Yaskawa INFORM job: pointsclTRJ4.JBI

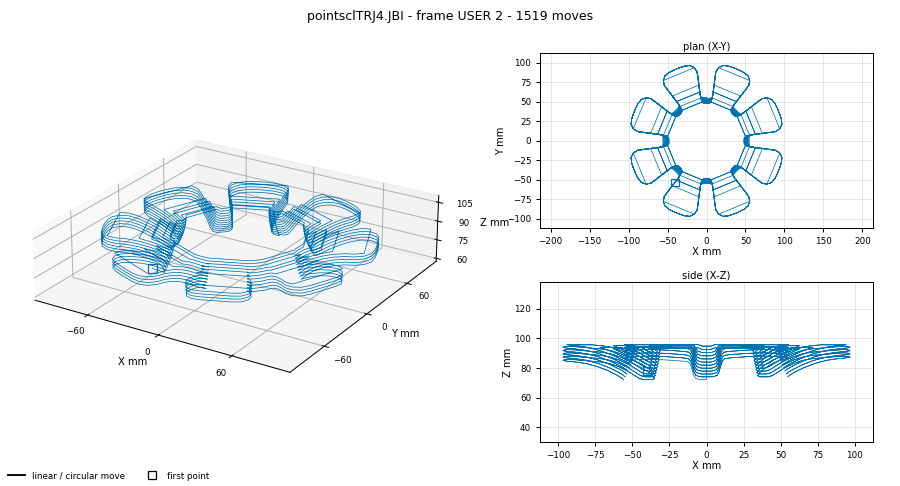
[picture p0: tool path of pointsclTRJ4.JBI in frame USER 2, 1519 of 1519 moves have a stored position in this frame; points joined in program order, loops and branches not executed]
/JOB
//NAME pointsclTRJ4
//POS
///NPOS 1519,0,0,0,0,0
///USER 2
///TOOL 1
///POSTYPE USER
///RECTAN
///RCONF 1,0,0,0,0,0,0,0,0,0,0,0,0,0,0,0,0,0,0,0,0,0,0,0
C00000=-40.007,-53.324,78.036,162.0773,27.0568,0.0000
C00001=-36.517,-48.718,75.143,159.1189,26.0241,0.0000
C00002=-35.037,-45.351,73.015,156.9441,24.9731,0.0000
C00003=-36.538,-42.505,72.166,153.8641,22.7812,0.0000
C00004=-38.303,-40.803,72.129,153.4120,22.4132,0.0000
C00005=-39.567,-39.567,72.154,154.3066,23.4380,0.0000
C00006=-40.803,-38.303,72.129,155.2410,24.4422,0.0000
C00007=-42.506,-36.538,72.166,154.9286,23.9614,0.0000
C00008=-45.352,-35.037,73.015,153.1527,20.7940,0.0000
C00009=-48.718,-36.517,75.143,152.4095,18.6805,0.0000
C00010=-53.324,-40.007,78.036,151.7719,15.9057,0.0000
C00011=-59.196,-44.618,80.927,152.7519,8.2885,0.0000
C00012=-65.578,-49.604,83.062,-179.3107,0.4201,0.0000
C00013=-71.524,-53.949,84.088,-176.3228,2.4871,0.0000
C00014=-77.795,-55.184,84.621,-175.2384,3.2785,0.0000
C00015=-83.601,-53.037,85.050,-174.7144,3.6343,0.0000
C00016=-87.741,-47.957,85.481,-174.6375,3.6773,0.0000
C00017=-90.934,-41.602,85.762,-174.7812,3.5713,0.0000
C00018=-93.717,-34.883,85.762,173.7849,-1.1544,0.0000
C00019=-95.953,-28.131,85.481,173.6084,-1.1802,0.0000
C00020=-96.617,-21.612,85.050,173.6932,-1.1566,0.0000
C00021=-94.030,-15.989,84.621,174.3152,-1.0407,0.0000
C00022=-88.723,-12.427,84.088,175.6413,-0.8379,0.0000
C00023=-81.446,-11.295,83.062,179.2156,-0.1904,0.0000
C00024=-73.408,-10.308,80.927,-166.0561,24.9794,0.0000
C00025=-65.995,-9.417,78.036,-171.4191,31.0262,0.0000
C00026=-60.270,-8.627,75.143,-174.3026,32.4608,0.0000
C00027=-56.844,-7.293,73.015,-176.7405,33.3374,0.0000
C00028=-55.892,-4.219,72.166,179.0738,34.1239,0.0000
C00029=-55.936,-1.768,72.129,178.4088,34.2068,0.0000
C00030=-55.957,0.000,72.154,179.9988,34.2310,0.0000
C00031=-55.936,1.767,72.129,-178.4074,34.2068,0.0000
C00032=-55.892,4.220,72.166,-179.0753,34.1238,0.0000
C00033=-56.844,7.293,73.015,176.7400,33.3374,0.0000
C00034=-60.270,8.627,75.143,174.3025,32.4608,0.0000
C00035=-65.995,9.417,78.036,171.4191,31.0263,0.0000
C00036=-73.408,10.308,80.927,166.0562,24.9798,0.0000
C00037=-81.446,11.295,83.062,-179.2156,-0.1904,0.0000
C00038=-88.723,12.427,84.088,-175.6413,-0.8379,0.0000
C00039=-94.030,15.989,84.621,-174.3152,-1.0407,0.0000
C00040=-96.617,21.612,85.050,-173.6932,-1.1566,0.0000
C00041=-95.953,28.131,85.481,-173.6084,-1.1802,0.0000
C00042=-93.717,34.883,85.762,-173.7849,-1.1544,0.0000
C00043=-90.934,41.602,85.762,174.7812,3.5713,0.0000
C00044=-87.741,47.957,85.481,174.6375,3.6773,0.0000
C00045=-83.601,53.037,85.050,174.7144,3.6343,0.0000
C00046=-77.795,55.184,84.621,175.2384,3.2785,0.0000
C00047=-71.524,53.949,84.088,176.3228,2.4871,0.0000
C00048=-65.578,49.604,83.062,179.3107,0.4201,0.0000
C00049=-59.196,44.618,80.927,-152.7521,8.2881,0.0000
C00050=-53.324,40.007,78.036,-151.7719,15.9056,0.0000
C00051=-48.718,36.517,75.143,-152.4095,18.6805,0.0000
C00052=-45.351,35.037,73.015,-153.1530,20.7943,0.0000
C00053=-42.505,36.538,72.166,-154.9295,23.9624,0.0000
C00054=-40.803,38.303,72.129,-155.2402,24.4413,0.0000
C00055=-39.567,39.567,72.154,-154.3081,23.4396,0.0000
C00056=-38.303,40.803,72.129,-153.4112,22.4123,0.0000
C00057=-36.538,42.506,72.166,-153.8651,22.7821,0.0000
C00058=-35.037,45.352,73.015,-156.9444,24.9734,0.0000
C00059=-36.517,48.718,75.143,-159.1190,26.0242,0.0000
C00060=-40.007,53.324,78.036,-162.0772,27.0569,0.0000
C00061=-44.618,59.196,80.927,-170.6940,26.9403,0.0000
C00062=-49.604,65.578,83.062,-179.5799,-0.6893,0.0000
C00063=-53.949,71.524,84.088,-177.5078,-3.6738,0.0000
C00064=-55.184,77.795,84.621,-176.7102,-4.7538,0.0000
C00065=-53.037,83.601,85.050,-176.3502,-5.2749,0.0000
C00066=-47.957,87.741,85.481,-176.3066,-5.3514,0.0000
C00067=-41.602,90.934,85.762,-176.4139,-5.2087,0.0000
C00068=-34.883,93.717,85.762,178.8388,6.2138,0.0000
C00069=-28.131,95.953,85.481,178.8125,6.3902,0.0000
C00070=-21.612,96.617,85.050,178.8363,6.3055,0.0000
C00071=-15.989,94.030,84.621,178.9542,5.6839,0.0000
C00072=-12.427,88.723,84.088,179.1597,4.3583,0.0000
C00073=-11.295,81.446,83.062,179.8096,0.7844,0.0000
C00074=-10.308,73.408,80.927,-154.3579,-12.6167,0.0000
C00075=-9.417,65.995,78.036,-148.6881,-7.3459,0.0000
C00076=-8.627,60.270,75.143,-147.4105,-4.8050,0.0000
C00077=-7.293,56.844,73.015,-146.6200,-2.7231,0.0000
C00078=-4.220,55.892,72.166,-145.8728,0.7655,0.0000
C00079=-1.767,55.936,72.129,-145.7829,1.3171,0.0000
C00080=0.000,55.957,72.154,-145.7690,-0.0010,0.0000
C00081=0.000,54.840,74.049,-146.5029,-0.0011,0.0000
C00082=1.666,54.823,74.024,-146.5152,-1.2504,0.0000
C00083=4.048,54.790,74.062,-146.6018,-0.7445,0.0000
C00084=7.088,55.804,74.943,-147.3459,2.7005,0.0000
C00085=8.393,59.388,77.145,-148.1466,4.7745,0.0000
C00086=9.180,65.335,80.122,-149.5349,7.4435,0.0000
C00087=10.089,72.980,83.074,-156.5768,13.0945,0.0000
C00088=11.094,81.206,85.240,179.6071,-1.7912,0.0000
C00089=12.226,88.613,86.276,179.1566,-4.6034,0.0000
C00090=15.808,94.009,86.813,178.9836,-5.7439,0.0000
C00091=21.475,96.642,87.246,178.8772,-6.3083,0.0000
C00092=28.048,95.980,87.679,178.8549,-6.3901,0.0000
C00093=34.856,93.728,87.962,178.8775,-6.2344,0.0000
C00094=41.629,90.922,87.962,-176.3720,5.1958,0.0000
C00095=48.035,87.701,87.679,-176.2769,5.3214,0.0000
C00096=53.151,83.521,87.246,-176.3195,5.2481,0.0000
C00097=55.296,77.652,86.813,-176.6467,4.7753,0.0000
C00098=54.014,71.304,86.276,-177.3359,3.8489,0.0000
C00099=49.577,65.266,85.240,-179.0109,1.5443,0.0000
C00100=44.470,58.738,83.074,-172.7574,-25.7204,0.0000
C00101=39.708,52.690,80.122,-162.8416,-26.5576,0.0000
C00102=36.059,47.928,77.145,-159.7054,-25.5142,0.0000
C00103=34.447,44.472,74.943,-157.5329,-24.4829,0.0000
C00104=35.880,41.605,74.062,-154.4883,-22.3343,0.0000
C00105=37.588,39.944,74.024,-154.0682,-21.9995,0.0000
C00106=38.778,38.778,74.049,-154.9210,-22.9691,0.0000
C00107=39.943,37.588,74.024,-155.8089,-23.9209,0.0000
C00108=41.605,35.880,74.062,-155.5235,-23.4763,0.0000
C00109=44.472,34.447,74.943,-153.7672,-20.3520,0.0000
C00110=47.928,36.059,77.145,-153.0297,-18.2415,0.0000
C00111=52.690,39.708,80.122,-152.3850,-15.3009,0.0000
C00112=58.738,44.470,83.074,-154.0994,-6.5221,0.0000
C00113=65.266,49.577,85.240,178.4555,-0.9887,0.0000
C00114=71.304,54.014,86.276,176.1470,-2.6581,0.0000
C00115=77.652,55.296,86.813,175.2165,-3.3416,0.0000
C00116=83.521,53.151,87.246,174.7411,-3.6651,0.0000
C00117=87.701,48.035,87.679,174.6674,-3.7070,0.0000
C00118=90.922,41.629,87.962,174.7939,-3.6131,0.0000
C00119=93.728,34.856,87.962,-173.7644,1.1158,0.0000
C00120=95.980,28.048,87.679,-173.6087,1.1380,0.0000
C00121=96.642,21.475,87.246,-173.6905,1.1160,0.0000
C00122=94.009,15.808,86.813,-174.2552,1.0113,0.0000
C00123=88.613,12.226,86.276,-175.3961,0.8406,0.0000
C00124=81.206,11.094,85.240,-178.2088,0.3927,0.0000
C00125=72.980,10.089,83.074,165.7755,-22.7793,0.0000
C00126=65.335,9.180,80.122,171.3809,-30.1815,0.0000
C00127=59.388,8.393,77.145,174.3839,-31.7299,0.0000
C00128=55.804,7.088,74.943,176.7935,-32.6133,0.0000
C00129=54.790,4.048,74.062,-179.1083,-33.3950,0.0000
C00130=54.823,1.666,74.024,-178.5009,-33.4758,0.0000
C00131=54.840,0.000,74.049,-179.9987,-33.4971,0.0000
C00132=54.823,-1.665,74.024,178.4994,-33.4758,0.0000
C00133=54.790,-4.048,74.062,179.1098,-33.3950,0.0000
C00134=55.804,-7.088,74.943,-176.7931,-32.6133,0.0000
C00135=59.388,-8.393,77.145,-174.3838,-31.7300,0.0000
C00136=65.335,-9.180,80.122,-171.3809,-30.1816,0.0000
C00137=72.980,-10.089,83.074,-165.7756,-22.7798,0.0000
C00138=81.206,-11.094,85.240,178.2088,0.3927,0.0000
C00139=88.613,-12.226,86.276,175.3961,0.8406,0.0000
C00140=94.009,-15.808,86.813,174.2552,1.0113,0.0000
C00141=96.642,-21.475,87.246,173.6905,1.1160,0.0000
C00142=95.980,-28.048,87.679,173.6087,1.1380,0.0000
C00143=93.728,-34.856,87.962,173.7644,1.1158,0.0000
C00144=90.922,-41.629,87.962,-174.7939,-3.6131,0.0000
C00145=87.701,-48.035,87.679,-174.6674,-3.7070,0.0000
C00146=83.521,-53.151,87.246,-174.7411,-3.6651,0.0000
C00147=77.652,-55.296,86.813,-175.2165,-3.3416,0.0000
C00148=71.304,-54.014,86.276,-176.1470,-2.6581,0.0000
C00149=65.266,-49.577,85.240,-178.4555,-0.9887,0.0000
C00150=58.738,-44.470,83.074,154.0997,-6.5217,0.0000
C00151=52.690,-39.708,80.122,152.3851,-15.3008,0.0000
C00152=47.928,-36.059,77.145,153.0298,-18.2415,0.0000
C00153=44.472,-34.447,74.943,153.7674,-20.3523,0.0000
C00154=41.605,-35.880,74.062,155.5243,-23.4773,0.0000
C00155=39.944,-37.588,74.024,155.8080,-23.9200,0.0000
C00156=38.778,-38.778,74.049,154.9225,-22.9708,0.0000
C00157=37.588,-39.943,74.024,154.0673,-21.9986,0.0000
C00158=35.880,-41.605,74.062,154.4893,-22.3352,0.0000
C00159=34.447,-44.472,74.943,157.5332,-24.4832,0.0000
C00160=36.059,-47.928,77.145,159.7054,-25.5143,0.0000
C00161=39.708,-52.690,80.122,162.8414,-26.5576,0.0000
C00162=44.470,-58.738,83.074,172.7569,-25.7206,0.0000
C00163=49.577,-65.266,85.240,179.0109,1.5443,0.0000
C00164=54.014,-71.304,86.276,177.3359,3.8489,0.0000
C00165=55.296,-77.652,86.813,176.6467,4.7753,0.0000
C00166=53.151,-83.521,87.246,176.3195,5.2481,0.0000
C00167=48.035,-87.701,87.679,176.2769,5.3214,0.0000
C00168=41.629,-90.922,87.962,176.3720,5.1958,0.0000
C00169=34.856,-93.728,87.962,-178.8775,-6.2344,0.0000
C00170=28.048,-95.980,87.679,-178.8549,-6.3901,0.0000
C00171=21.475,-96.642,87.246,-178.8772,-6.3083,0.0000
C00172=15.808,-94.009,86.813,-178.9836,-5.7439,0.0000
C00173=12.226,-88.613,86.276,-179.1566,-4.6034,0.0000
C00174=11.094,-81.206,85.240,-179.6071,-1.7912,0.0000
C00175=10.089,-72.980,83.074,156.5768,13.0945,0.0000
C00176=9.180,-65.335,80.122,149.5349,7.4435,0.0000
C00177=8.393,-59.388,77.145,148.1466,4.7745,0.0000
C00178=7.088,-55.804,74.943,147.3459,2.7005,0.0000
C00179=4.048,-54.790,74.062,146.6018,-0.7445,0.0000
C00180=1.666,-54.823,74.024,146.5152,-1.2504,0.0000
C00181=0.000,-54.840,74.049,146.5029,-0.0011,0.0000
C00182=0.000,-54.840,74.049,146.5029,-0.0011,0.0000
C00183=-1.665,-54.823,74.024,146.5152,1.2517,0.0000
C00184=-4.048,-54.790,74.062,146.6019,0.7432,0.0000
C00185=-7.088,-55.804,74.943,147.3460,-2.7009,0.0000
C00186=-8.393,-59.388,77.145,148.1466,-4.7746,0.0000
C00187=-9.180,-65.335,80.122,149.5348,-7.4435,0.0000
C00188=-10.089,-72.980,83.074,156.5763,-13.0943,0.0000
C00189=-11.094,-81.206,85.240,-179.6071,1.7912,0.0000
C00190=-12.226,-88.613,86.276,-179.1566,4.6034,0.0000
C00191=-15.808,-94.009,86.813,-178.9836,5.7439,0.0000
C00192=-21.475,-96.642,87.246,-178.8772,6.3083,0.0000
C00193=-28.048,-95.980,87.679,-178.8549,6.3901,0.0000
C00194=-34.856,-93.728,87.962,-178.8775,6.2344,0.0000
C00195=-41.629,-90.922,87.962,176.3720,-5.1958,0.0000
C00196=-48.035,-87.701,87.679,176.2769,-5.3214,0.0000
C00197=-53.151,-83.521,87.246,176.3195,-5.2481,0.0000
C00198=-55.296,-77.652,86.813,176.6467,-4.7753,0.0000
C00199=-54.014,-71.304,86.276,177.3359,-3.8489,0.0000
C00200=-49.577,-65.266,85.240,179.0109,-1.5443,0.0000
C00201=-44.470,-58.738,83.074,172.7574,25.7204,0.0000
C00202=-39.708,-52.690,80.122,162.8416,26.5576,0.0000
C00203=-36.059,-47.928,77.145,159.7054,25.5142,0.0000
C00204=-34.447,-44.472,74.943,157.5329,24.4829,0.0000
C00205=-35.880,-41.605,74.062,154.4883,22.3343,0.0000
C00206=-37.588,-39.944,74.024,154.0682,21.9995,0.0000
C00207=-38.778,-38.778,74.049,154.9210,22.9691,0.0000
C00208=-39.943,-37.588,74.024,155.8089,23.9209,0.0000
C00209=-41.605,-35.880,74.062,155.5235,23.4763,0.0000
C00210=-44.472,-34.447,74.943,153.7672,20.3520,0.0000
C00211=-47.928,-36.059,77.145,153.0297,18.2415,0.0000
C00212=-52.690,-39.708,80.122,152.3850,15.3009,0.0000
C00213=-58.738,-44.470,83.074,154.0994,6.5221,0.0000
C00214=-65.266,-49.577,85.240,-178.4555,0.9887,0.0000
C00215=-71.304,-54.014,86.276,-176.1470,2.6581,0.0000
C00216=-77.652,-55.296,86.813,-175.2165,3.3416,0.0000
C00217=-83.521,-53.151,87.246,-174.7411,3.6651,0.0000
C00218=-87.701,-48.035,87.679,-174.6674,3.7070,0.0000
C00219=-90.922,-41.629,87.962,-174.7939,3.6131,0.0000
C00220=-93.728,-34.856,87.962,173.7644,-1.1158,0.0000
C00221=-95.980,-28.048,87.679,173.6087,-1.1380,0.0000
C00222=-96.642,-21.475,87.246,173.6905,-1.1160,0.0000
C00223=-94.009,-15.808,86.813,174.2552,-1.0113,0.0000
C00224=-88.613,-12.226,86.276,175.3961,-0.8406,0.0000
C00225=-81.206,-11.094,85.240,178.2088,-0.3927,0.0000
C00226=-72.980,-10.089,83.074,-165.7755,22.7793,0.0000
C00227=-65.335,-9.180,80.122,-171.3809,30.1815,0.0000
C00228=-59.388,-8.393,77.145,-174.3839,31.7299,0.0000
C00229=-55.804,-7.088,74.943,-176.7935,32.6133,0.0000
C00230=-54.790,-4.048,74.062,179.1083,33.3950,0.0000
C00231=-54.823,-1.666,74.024,178.5009,33.4758,0.0000
C00232=-54.840,0.000,74.049,179.9987,33.4971,0.0000
C00233=-54.823,1.665,74.024,-178.4994,33.4758,0.0000
C00234=-54.790,4.048,74.062,-179.1098,33.3950,0.0000
C00235=-55.804,7.088,74.943,176.7931,32.6133,0.0000
C00236=-59.388,8.393,77.145,174.3838,31.7300,0.0000
C00237=-65.335,9.180,80.122,171.3809,30.1816,0.0000
C00238=-72.980,10.089,83.074,165.7756,22.7798,0.0000
C00239=-81.206,11.094,85.240,-178.2088,-0.3927,0.0000
C00240=-88.613,12.226,86.276,-175.3961,-0.8406,0.0000
C00241=-94.009,15.808,86.813,-174.2552,-1.0113,0.0000
C00242=-96.642,21.475,87.246,-173.6905,-1.1160,0.0000
C00243=-95.980,28.048,87.679,-173.6087,-1.1380,0.0000
C00244=-93.728,34.856,87.962,-173.7644,-1.1158,0.0000
C00245=-90.922,41.629,87.962,174.7939,3.6131,0.0000
C00246=-87.701,48.035,87.679,174.6674,3.7070,0.0000
C00247=-83.521,53.151,87.246,174.7411,3.6651,0.0000
C00248=-77.652,55.296,86.813,175.2165,3.3416,0.0000
C00249=-71.304,54.014,86.276,176.1470,2.6581,0.0000
C00250=-65.266,49.577,85.240,178.4555,0.9887,0.0000
C00251=-58.738,44.470,83.074,-154.0997,6.5217,0.0000
C00252=-52.690,39.708,80.122,-152.3851,15.3008,0.0000
C00253=-47.928,36.059,77.145,-153.0298,18.2415,0.0000
C00254=-44.472,34.447,74.943,-153.7674,20.3523,0.0000
C00255=-41.605,35.880,74.062,-155.5243,23.4773,0.0000
C00256=-39.944,37.588,74.024,-155.8080,23.9200,0.0000
C00257=-38.778,38.778,74.049,-154.9225,22.9708,0.0000
C00258=-37.588,39.943,74.024,-154.0673,21.9986,0.0000
C00259=-35.880,41.605,74.062,-154.4893,22.3352,0.0000
C00260=-34.447,44.472,74.943,-157.5332,24.4832,0.0000
C00261=-36.059,47.928,77.145,-159.7054,25.5143,0.0000
C00262=-39.708,52.690,80.122,-162.8414,26.5576,0.0000
C00263=-44.470,58.738,83.074,-172.7569,25.7206,0.0000
C00264=-49.577,65.266,85.240,-179.0109,-1.5443,0.0000
C00265=-54.014,71.304,86.276,-177.3359,-3.8489,0.0000
C00266=-55.296,77.652,86.813,-176.6467,-4.7753,0.0000
C00267=-53.151,83.521,87.246,-176.3195,-5.2481,0.0000
C00268=-48.035,87.701,87.679,-176.2769,-5.3214,0.0000
C00269=-41.629,90.922,87.962,-176.3720,-5.1958,0.0000
C00270=-34.856,93.728,87.962,178.8775,6.2344,0.0000
C00271=-28.048,95.980,87.679,178.8549,6.3901,0.0000
C00272=-21.475,96.642,87.246,178.8772,6.3083,0.0000
C00273=-15.808,94.009,86.813,178.9836,5.7439,0.0000
C00274=-12.226,88.613,86.276,179.1566,4.6034,0.0000
C00275=-11.094,81.206,85.240,179.6071,1.7912,0.0000
C00276=-10.089,72.980,83.074,-156.5763,-13.0943,0.0000
C00277=-9.180,65.335,80.122,-149.5348,-7.4435,0.0000
C00278=-8.393,59.388,77.145,-148.1466,-4.7746,0.0000
C00279=-7.088,55.804,74.943,-147.3460,-2.7009,0.0000
C00280=-4.048,54.790,74.062,-146.6019,0.7432,0.0000
C00281=-1.665,54.823,74.024,-146.5152,1.2517,0.0000
C00282=0.000,54.840,74.049,-146.5029,-0.0011,0.0000
C00283=0.000,53.776,75.975,-147.2942,-0.0011,0.0000
C00284=1.568,53.762,75.948,-147.3046,-1.1830,0.0000
C00285=3.884,53.739,75.988,-147.3883,-0.7211,0.0000
C00286=6.894,54.818,76.900,-148.1310,2.6757,0.0000
C00287=8.175,58.565,79.173,-148.9497,4.7476,0.0000
C00288=8.965,64.737,82.228,-150.4833,7.5652,0.0000
C00289=9.898,72.606,85.234,-159.4646,13.4583,0.0000
C00290=10.924,81.005,87.424,179.4966,-2.4962,0.0000
C00291=12.061,88.524,88.468,179.1698,-4.7418,0.0000
C00292=15.662,93.991,89.008,179.0218,-5.7312,0.0000
C00293=21.365,96.662,89.443,178.9256,-6.2465,0.0000
C00294=27.983,96.002,89.878,178.9048,-6.3264,0.0000
C00295=34.834,93.736,90.162,178.9241,-6.1910,0.0000
C00296=41.650,90.913,90.162,-176.3701,5.1323,0.0000
C00297=48.097,87.670,89.878,-176.2872,5.2413,0.0000
C00298=53.243,83.458,89.443,-176.3295,5.1704,0.0000
C00299=55.387,77.537,89.008,-176.6290,4.7394,0.0000
C00300=54.067,71.124,88.468,-177.2282,3.9373,0.0000
C00301=49.554,65.004,87.424,-178.5900,2.1207,0.0000
C00302=44.341,58.339,85.234,-175.1885,-23.9414,0.0000
C00303=39.437,52.115,82.228,-163.7002,-26.0042,0.0000
C00304=35.631,47.192,79.173,-160.3448,-24.9604,0.0000
C00305=33.888,43.637,76.900,-158.1643,-23.9500,0.0000
C00306=35.253,40.746,75.988,-155.1567,-21.8490,0.0000
C00307=36.906,39.124,75.948,-154.7690,-21.5479,0.0000
C00308=38.025,38.025,75.975,-155.5786,-22.4610,0.0000
C00309=39.124,36.906,75.948,-156.4186,-23.3591,0.0000
C00310=40.746,35.253,75.988,-156.1608,-22.9509,0.0000
C00311=43.637,33.888,76.901,-154.4279,-19.8718,0.0000
C00312=47.192,35.631,79.173,-153.6983,-17.7547,0.0000
C00313=52.115,39.437,82.228,-153.0579,-14.6108,0.0000
C00314=58.339,44.341,85.234,-155.9831,-4.3971,0.0000
C00315=65.004,49.554,87.424,177.8787,-1.4090,0.0000
C00316=71.124,54.067,88.468,176.0581,-2.7652,0.0000
C00317=77.537,55.387,89.008,175.2524,-3.3595,0.0000
C00318=83.458,53.243,89.443,174.8190,-3.6556,0.0000
C00319=87.670,48.097,89.878,174.7477,-3.6973,0.0000
C00320=90.913,41.650,90.162,174.8574,-3.6153,0.0000
C00321=93.736,34.834,90.162,-173.8080,1.0696,0.0000
C00322=96.002,27.983,89.878,-173.6725,1.0885,0.0000
C00323=96.662,21.365,89.443,-173.7524,1.0680,0.0000
C00324=93.991,15.662,89.008,-174.2680,0.9733,0.0000
C00325=88.524,12.061,88.468,-175.2577,0.8274,0.0000
C00326=81.005,10.924,87.424,-177.5037,0.5030,0.0000
C00327=72.606,9.898,85.234,165.6649,-19.9471,0.0000
C00328=64.737,8.965,82.228,171.3226,-29.2348,0.0000
C00329=58.565,8.175,79.173,174.4630,-30.9320,0.0000
C00330=54.818,6.894,76.900,176.8503,-31.8302,0.0000
C00331=53.739,3.884,75.988,-179.1440,-32.6088,0.0000
C00332=53.762,1.568,75.948,-178.5943,-32.6875,0.0000
C00333=53.776,0.000,75.975,-179.9987,-32.7058,0.0000
C00334=53.762,-1.568,75.948,178.5928,-32.6875,0.0000
C00335=53.739,-3.885,75.988,179.1455,-32.6088,0.0000
C00336=54.819,-6.894,76.901,-176.8499,-31.8301,0.0000
C00337=58.565,-8.175,79.173,-174.4629,-30.9321,0.0000
C00338=64.737,-8.965,82.228,-171.3226,-29.2349,0.0000
C00339=72.606,-9.898,85.234,-165.6650,-19.9477,0.0000
C00340=81.005,-10.924,87.424,177.5037,0.5030,0.0000
C00341=88.524,-12.061,88.468,175.2577,0.8274,0.0000
C00342=93.991,-15.662,89.008,174.2680,0.9733,0.0000
C00343=96.662,-21.365,89.443,173.7524,1.0680,0.0000
C00344=96.002,-27.983,89.878,173.6725,1.0885,0.0000
C00345=93.736,-34.834,90.162,173.8080,1.0696,0.0000
C00346=90.913,-41.650,90.162,-174.8574,-3.6153,0.0000
C00347=87.670,-48.097,89.878,-174.7477,-3.6973,0.0000
C00348=83.458,-53.243,89.443,-174.8190,-3.6556,0.0000
C00349=77.537,-55.387,89.008,-175.2524,-3.3595,0.0000
C00350=71.124,-54.067,88.468,-176.0581,-2.7652,0.0000
C00351=65.004,-49.554,87.424,-177.8787,-1.4090,0.0000
C00352=58.339,-44.341,85.234,155.9835,-4.3966,0.0000
C00353=52.115,-39.437,82.228,153.0580,-14.6107,0.0000
C00354=47.192,-35.631,79.173,153.6984,-17.7548,0.0000
C00355=43.637,-33.888,76.900,154.4281,-19.8721,0.0000
C00356=40.746,-35.253,75.988,156.1616,-22.9519,0.0000
C00357=39.124,-36.906,75.948,156.4177,-23.3581,0.0000
C00358=38.025,-38.025,75.975,155.5800,-22.4627,0.0000
C00359=36.906,-39.124,75.948,154.7681,-21.5469,0.0000
C00360=35.253,-40.746,75.988,155.1576,-21.8499,0.0000
C00361=33.888,-43.637,76.901,158.1646,-23.9503,0.0000
C00362=35.631,-47.192,79.173,160.3448,-24.9605,0.0000
C00363=39.437,-52.115,82.228,163.7000,-26.0042,0.0000
C00364=44.341,-58.339,85.234,175.1880,-23.9418,0.0000
C00365=49.554,-65.004,87.424,178.5900,2.1207,0.0000
C00366=54.067,-71.124,88.468,177.2282,3.9373,0.0000
C00367=55.387,-77.537,89.008,176.6290,4.7394,0.0000
C00368=53.243,-83.458,89.443,176.3295,5.1704,0.0000
C00369=48.097,-87.670,89.878,176.2872,5.2413,0.0000
C00370=41.650,-90.913,90.162,176.3701,5.1323,0.0000
C00371=34.834,-93.736,90.162,-178.9241,-6.1910,0.0000
C00372=27.983,-96.002,89.878,-178.9048,-6.3264,0.0000
C00373=21.365,-96.662,89.443,-178.9256,-6.2465,0.0000
C00374=15.662,-93.991,89.008,-179.0218,-5.7312,0.0000
C00375=12.061,-88.524,88.468,-179.1698,-4.7418,0.0000
C00376=10.924,-81.005,87.424,-179.4966,-2.4962,0.0000
C00377=9.898,-72.606,85.234,159.4646,13.4583,0.0000
C00378=8.965,-64.737,82.228,150.4833,7.5652,0.0000
C00379=8.175,-58.565,79.173,148.9497,4.7476,0.0000
C00380=6.894,-54.818,76.900,148.1310,2.6757,0.0000
C00381=3.884,-53.739,75.988,147.3883,-0.7211,0.0000
C00382=1.568,-53.762,75.948,147.3046,-1.1830,0.0000
C00383=0.000,-53.776,75.975,147.2942,-0.0011,0.0000
C00384=0.000,-53.776,75.975,147.2942,-0.0011,0.0000
C00385=-1.568,-53.762,75.948,147.3046,1.1843,0.0000
C00386=-3.885,-53.739,75.988,147.3883,0.7198,0.0000
C00387=-6.894,-54.819,76.901,148.1310,-2.6760,0.0000
C00388=-8.175,-58.565,79.173,148.9496,-4.7476,0.0000
C00389=-8.965,-64.737,82.228,150.4831,-7.5651,0.0000
C00390=-9.898,-72.606,85.234,159.4640,-13.4582,0.0000
C00391=-10.924,-81.005,87.424,-179.4966,2.4962,0.0000
C00392=-12.061,-88.524,88.468,-179.1698,4.7418,0.0000
C00393=-15.662,-93.991,89.008,-179.0218,5.7312,0.0000
C00394=-21.365,-96.662,89.443,-178.9256,6.2465,0.0000
C00395=-27.983,-96.002,89.878,-178.9048,6.3264,0.0000
C00396=-34.834,-93.736,90.162,-178.9241,6.1910,0.0000
C00397=-41.650,-90.913,90.162,176.3701,-5.1323,0.0000
C00398=-48.097,-87.670,89.878,176.2872,-5.2413,0.0000
C00399=-53.243,-83.458,89.443,176.3295,-5.1704,0.0000
C00400=-55.387,-77.537,89.008,176.6290,-4.7394,0.0000
C00401=-54.067,-71.124,88.468,177.2282,-3.9373,0.0000
C00402=-49.554,-65.004,87.424,178.5900,-2.1207,0.0000
C00403=-44.341,-58.339,85.234,175.1885,23.9414,0.0000
C00404=-39.437,-52.115,82.228,163.7002,26.0042,0.0000
C00405=-35.631,-47.192,79.173,160.3448,24.9604,0.0000
C00406=-33.888,-43.637,76.900,158.1643,23.9500,0.0000
C00407=-35.253,-40.746,75.988,155.1567,21.8490,0.0000
C00408=-36.906,-39.124,75.948,154.7690,21.5479,0.0000
C00409=-38.025,-38.025,75.975,155.5786,22.4610,0.0000
C00410=-39.124,-36.906,75.948,156.4186,23.3591,0.0000
C00411=-40.746,-35.253,75.988,156.1608,22.9509,0.0000
C00412=-43.637,-33.888,76.901,154.4279,19.8718,0.0000
C00413=-47.192,-35.631,79.173,153.6983,17.7547,0.0000
C00414=-52.115,-39.437,82.228,153.0579,14.6108,0.0000
C00415=-58.339,-44.341,85.234,155.9831,4.3971,0.0000
C00416=-65.004,-49.554,87.424,-177.8787,1.4090,0.0000
C00417=-71.124,-54.067,88.468,-176.0581,2.7652,0.0000
C00418=-77.537,-55.387,89.008,-175.2524,3.3595,0.0000
C00419=-83.458,-53.243,89.443,-174.8190,3.6556,0.0000
C00420=-87.670,-48.097,89.878,-174.7477,3.6973,0.0000
C00421=-90.913,-41.650,90.162,-174.8574,3.6153,0.0000
C00422=-93.736,-34.834,90.162,173.8080,-1.0696,0.0000
C00423=-96.002,-27.983,89.878,173.6725,-1.0885,0.0000
C00424=-96.662,-21.365,89.443,173.7524,-1.0680,0.0000
C00425=-93.991,-15.662,89.008,174.2680,-0.9733,0.0000
C00426=-88.524,-12.061,88.468,175.2577,-0.8274,0.0000
C00427=-81.005,-10.924,87.424,177.5037,-0.5030,0.0000
C00428=-72.606,-9.898,85.234,-165.6649,19.9471,0.0000
C00429=-64.737,-8.965,82.228,-171.3226,29.2348,0.0000
C00430=-58.565,-8.175,79.173,-174.4630,30.9320,0.0000
C00431=-54.818,-6.894,76.900,-176.8503,31.8302,0.0000
C00432=-53.739,-3.884,75.988,179.1440,32.6088,0.0000
C00433=-53.762,-1.568,75.948,178.5943,32.6875,0.0000
C00434=-53.776,0.000,75.975,179.9987,32.7058,0.0000
C00435=-53.762,1.568,75.948,-178.5928,32.6875,0.0000
C00436=-53.739,3.885,75.988,-179.1455,32.6088,0.0000
C00437=-54.819,6.894,76.901,176.8499,31.8301,0.0000
C00438=-58.565,8.175,79.173,174.4629,30.9321,0.0000
C00439=-64.737,8.965,82.228,171.3226,29.2349,0.0000
C00440=-72.606,9.898,85.234,165.6650,19.9477,0.0000
C00441=-81.005,10.924,87.424,-177.5037,-0.5030,0.0000
C00442=-88.524,12.061,88.468,-175.2577,-0.8274,0.0000
C00443=-93.991,15.662,89.008,-174.2680,-0.9733,0.0000
C00444=-96.662,21.365,89.443,-173.7524,-1.0680,0.0000
C00445=-96.002,27.983,89.878,-173.6725,-1.0885,0.0000
C00446=-93.736,34.834,90.162,-173.8080,-1.0696,0.0000
C00447=-90.913,41.650,90.162,174.8574,3.6153,0.0000
C00448=-87.670,48.097,89.878,174.7477,3.6973,0.0000
C00449=-83.458,53.243,89.443,174.8190,3.6556,0.0000
C00450=-77.537,55.387,89.008,175.2524,3.3595,0.0000
C00451=-71.124,54.067,88.468,176.0581,2.7652,0.0000
C00452=-65.004,49.554,87.424,177.8787,1.4090,0.0000
C00453=-58.339,44.341,85.234,-155.9835,4.3966,0.0000
C00454=-52.115,39.437,82.228,-153.0580,14.6107,0.0000
C00455=-47.192,35.631,79.173,-153.6984,17.7548,0.0000
C00456=-43.637,33.888,76.900,-154.4281,19.8721,0.0000
C00457=-40.746,35.253,75.988,-156.1616,22.9519,0.0000
C00458=-39.124,36.906,75.948,-156.4177,23.3581,0.0000
C00459=-38.025,38.025,75.975,-155.5800,22.4627,0.0000
C00460=-36.906,39.124,75.948,-154.7681,21.5469,0.0000
C00461=-35.253,40.746,75.988,-155.1576,21.8499,0.0000
C00462=-33.888,43.637,76.901,-158.1646,23.9503,0.0000
C00463=-35.631,47.192,79.173,-160.3448,24.9605,0.0000
C00464=-39.437,52.115,82.228,-163.7000,26.0042,0.0000
C00465=-44.341,58.339,85.234,-175.1880,23.9418,0.0000
C00466=-49.554,65.004,87.424,-178.5900,-2.1207,0.0000
C00467=-54.067,71.124,88.468,-177.2282,-3.9373,0.0000
C00468=-55.387,77.537,89.008,-176.6290,-4.7394,0.0000
C00469=-53.243,83.458,89.443,-176.3295,-5.1704,0.0000
C00470=-48.097,87.670,89.878,-176.2872,-5.2413,0.0000
C00471=-41.650,90.913,90.162,-176.3701,-5.1323,0.0000
C00472=-34.834,93.736,90.162,178.9241,6.1910,0.0000
C00473=-27.983,96.002,89.878,178.9048,6.3264,0.0000
C00474=-21.365,96.662,89.443,178.9256,6.2465,0.0000
C00475=-15.662,93.991,89.008,179.0218,5.7312,0.0000
C00476=-12.061,88.524,88.468,179.1698,4.7418,0.0000
C00477=-10.924,81.005,87.424,179.4966,2.4962,0.0000
C00478=-9.898,72.606,85.234,-159.4640,-13.4582,0.0000
C00479=-8.965,64.737,82.228,-150.4831,-7.5651,0.0000
C00480=-8.175,58.565,79.173,-148.9496,-4.7476,0.0000
C00481=-6.894,54.819,76.901,-148.1310,-2.6760,0.0000
C00482=-3.885,53.739,75.988,-147.3883,0.7198,0.0000
C00483=-1.568,53.762,75.948,-147.3046,1.1843,0.0000
C00484=0.000,53.776,75.975,-147.2942,-0.0011,0.0000
C00485=0.000,52.771,77.932,-148.1446,-0.0011,0.0000
C00486=1.476,52.759,77.904,-148.1532,-1.1142,0.0000
C00487=3.730,52.747,77.945,-148.2340,-0.6953,0.0000
C00488=6.711,53.894,78.888,-148.9777,2.6500,0.0000
C00489=7.974,57.808,81.229,-149.8240,4.7265,0.0000
C00490=8.774,64.206,84.354,-151.5479,7.7153,0.0000
C00491=9.737,72.291,87.405,-163.2875,13.4370,0.0000
C00492=10.790,80.844,89.614,179.4406,-2.9775,0.0000
C00493=11.935,88.455,90.663,179.1947,-4.7897,0.0000
C00494=15.553,93.978,91.206,179.0669,-5.6522,0.0000
C00495=21.285,96.677,91.642,178.9803,-6.1239,0.0000
C00496=27.936,96.017,92.077,178.9611,-6.2020,0.0000
C00497=34.820,93.742,92.362,178.9774,-6.0859,0.0000
C00498=41.664,90.907,92.362,-176.4075,5.0207,0.0000
C00499=48.140,87.648,92.077,-176.3363,5.1140,0.0000
C00500=53.310,83.412,91.642,-176.3785,5.0454,0.0000
C00501=55.455,77.451,91.206,-176.6534,4.6520,0.0000
C00502=54.108,70.986,90.663,-177.1767,3.9534,0.0000
C00503=49.536,64.795,89.614,-178.2887,2.5002,0.0000
C00504=44.233,58.003,87.405,-177.9428,-21.2286,0.0000
C00505=39.197,51.604,84.354,-164.6661,-25.3891,0.0000
C00506=35.238,46.514,81.229,-161.0413,-24.3614,0.0000
C00507=33.363,42.854,78.888,-158.8407,-23.3737,0.0000
C00508=34.660,39.935,77.945,-155.8706,-21.3245,0.0000
C00509=36.262,38.350,77.904,-155.5148,-21.0563,0.0000
C00510=37.314,37.314,77.932,-156.2799,-21.9120,0.0000
C00511=38.350,36.262,77.904,-157.0708,-22.7556,0.0000
C00512=39.935,34.660,77.945,-156.8403,-22.3829,0.0000
C00513=42.854,33.363,78.888,-155.1350,-19.3498,0.0000
C00514=46.514,35.238,81.229,-154.4158,-17.2150,0.0000
C00515=51.604,39.197,84.354,-153.7972,-13.8220,0.0000
C00516=58.003,44.233,87.405,-158.7585,-1.9180,0.0000
C00517=64.795,49.536,89.614,177.4986,-1.7097,0.0000
C00518=70.986,54.108,90.663,176.0418,-2.8166,0.0000
C00519=77.451,55.455,91.206,175.3401,-3.3356,0.0000
C00520=83.412,53.310,91.642,174.9446,-3.6075,0.0000
C00521=87.648,48.140,92.077,174.8756,-3.6491,0.0000
C00522=90.907,41.664,92.362,174.9695,-3.5787,0.0000
C00523=93.742,34.820,92.362,-173.9131,1.0168,0.0000
C00524=96.017,27.936,92.077,-173.7970,1.0328,0.0000
C00525=96.677,21.285,91.642,-173.8752,1.0139,0.0000
C00526=93.978,15.553,91.206,-174.3470,0.9286,0.0000
C00527=88.455,11.935,90.663,-175.2098,0.8024,0.0000
C00528=80.844,10.790,89.614,-177.0224,0.5586,0.0000
C00529=72.291,9.737,87.405,165.9933,-16.2421,0.0000
C00530=64.206,8.774,84.354,171.2402,-28.1714,0.0000
C00531=57.808,7.974,81.229,174.5367,-30.0628,0.0000
C00532=53.894,6.711,78.888,176.9085,-30.9855,0.0000
C00533=52.747,3.730,77.945,-179.1822,-31.7634,0.0000
C00534=52.759,1.476,77.904,-178.6884,-31.8401,0.0000
C00535=52.771,0.000,77.932,-179.9987,-31.8554,0.0000
C00536=52.759,-1.476,77.904,178.6868,-31.8401,0.0000
C00537=52.747,-3.730,77.945,179.1836,-31.7633,0.0000
C00538=53.894,-6.711,78.888,-176.9080,-30.9854,0.0000
C00539=57.808,-7.974,81.229,-174.5367,-30.0629,0.0000
C00540=64.206,-8.774,84.354,-171.2403,-28.1716,0.0000
C00541=72.291,-9.737,87.405,-165.9932,-16.2427,0.0000
C00542=80.844,-10.790,89.614,177.0224,0.5586,0.0000
C00543=88.455,-11.935,90.663,175.2098,0.8024,0.0000
C00544=93.978,-15.553,91.206,174.3470,0.9286,0.0000
C00545=96.677,-21.285,91.642,173.8752,1.0139,0.0000
C00546=96.017,-27.936,92.077,173.7970,1.0328,0.0000
C00547=93.742,-34.820,92.362,173.9131,1.0168,0.0000
C00548=90.907,-41.664,92.362,-174.9695,-3.5787,0.0000
C00549=87.648,-48.140,92.077,-174.8756,-3.6491,0.0000
C00550=83.412,-53.310,91.642,-174.9446,-3.6075,0.0000
C00551=77.451,-55.455,91.206,-175.3401,-3.3356,0.0000
C00552=70.986,-54.108,90.663,-176.0418,-2.8166,0.0000
C00553=64.795,-49.536,89.614,-177.4986,-1.7097,0.0000
C00554=58.003,-44.233,87.405,158.7589,-1.9176,0.0000
C00555=51.604,-39.197,84.354,153.7973,-13.8218,0.0000
C00556=46.514,-35.238,81.229,154.4159,-17.2150,0.0000
C00557=42.854,-33.363,78.888,155.1352,-19.3501,0.0000
C00558=39.935,-34.660,77.945,156.8411,-22.3839,0.0000
C00559=38.350,-36.262,77.904,157.0699,-22.7546,0.0000
C00560=37.314,-37.314,77.932,156.2814,-21.9136,0.0000
C00561=36.262,-38.350,77.904,155.5138,-21.0553,0.0000
C00562=34.660,-39.935,77.945,155.8715,-21.3254,0.0000
C00563=33.363,-42.854,78.888,158.8410,-23.3739,0.0000
C00564=35.238,-46.514,81.229,161.0413,-24.3614,0.0000
C00565=39.197,-51.604,84.354,164.6659,-25.3892,0.0000
C00566=44.233,-58.003,87.405,177.9423,-21.2290,0.0000
C00567=49.536,-64.795,89.614,178.2887,2.5002,0.0000
C00568=54.108,-70.986,90.663,177.1767,3.9534,0.0000
C00569=55.455,-77.451,91.206,176.6534,4.6520,0.0000
C00570=53.310,-83.412,91.642,176.3785,5.0454,0.0000
C00571=48.140,-87.648,92.077,176.3363,5.1140,0.0000
C00572=41.664,-90.907,92.362,176.4075,5.0207,0.0000
C00573=34.820,-93.742,92.362,-178.9774,-6.0859,0.0000
C00574=27.936,-96.017,92.077,-178.9611,-6.2020,0.0000
C00575=21.285,-96.677,91.642,-178.9803,-6.1239,0.0000
C00576=15.553,-93.978,91.206,-179.0669,-5.6522,0.0000
C00577=11.935,-88.455,90.663,-179.1947,-4.7897,0.0000
C00578=10.790,-80.844,89.614,-179.4406,-2.9775,0.0000
C00579=9.737,-72.291,87.405,163.2875,13.4370,0.0000
C00580=8.774,-64.206,84.354,151.5479,7.7153,0.0000
C00581=7.974,-57.808,81.229,149.8240,4.7265,0.0000
C00582=6.711,-53.894,78.888,148.9777,2.6500,0.0000
C00583=3.730,-52.747,77.945,148.2340,-0.6953,0.0000
C00584=1.476,-52.759,77.904,148.1532,-1.1142,0.0000
C00585=0.000,-52.771,77.932,148.1446,-0.0011,0.0000
C00586=0.000,-52.771,77.932,148.1446,-0.0011,0.0000
C00587=-1.476,-52.759,77.904,148.1532,1.1155,0.0000
C00588=-3.730,-52.747,77.945,148.2341,0.6941,0.0000
C00589=-6.711,-53.894,78.888,148.9777,-2.6504,0.0000
C00590=-7.974,-57.808,81.229,149.8239,-4.7266,0.0000
C00591=-8.774,-64.206,84.354,151.5477,-7.7153,0.0000
C00592=-9.737,-72.291,87.405,163.2869,-13.4370,0.0000
C00593=-10.790,-80.844,89.614,-179.4406,2.9775,0.0000
C00594=-11.935,-88.455,90.663,-179.1947,4.7897,0.0000
C00595=-15.553,-93.978,91.206,-179.0669,5.6522,0.0000
C00596=-21.285,-96.677,91.642,-178.9803,6.1239,0.0000
C00597=-27.936,-96.017,92.077,-178.9611,6.2020,0.0000
C00598=-34.820,-93.742,92.362,-178.9774,6.0859,0.0000
C00599=-41.664,-90.907,92.362,176.4075,-5.0207,0.0000
C00600=-48.140,-87.648,92.077,176.3363,-5.1140,0.0000
C00601=-53.310,-83.412,91.642,176.3785,-5.0454,0.0000
C00602=-55.455,-77.451,91.206,176.6534,-4.6520,0.0000
C00603=-54.108,-70.986,90.663,177.1767,-3.9534,0.0000
C00604=-49.536,-64.795,89.614,178.2887,-2.5002,0.0000
C00605=-44.233,-58.003,87.405,177.9428,21.2286,0.0000
C00606=-39.197,-51.604,84.354,164.6661,25.3891,0.0000
C00607=-35.238,-46.514,81.229,161.0413,24.3614,0.0000
C00608=-33.363,-42.854,78.888,158.8407,23.3737,0.0000
C00609=-34.660,-39.935,77.945,155.8706,21.3245,0.0000
C00610=-36.262,-38.350,77.904,155.5148,21.0563,0.0000
C00611=-37.314,-37.314,77.932,156.2799,21.9120,0.0000
C00612=-38.350,-36.262,77.904,157.0708,22.7556,0.0000
C00613=-39.935,-34.660,77.945,156.8403,22.3829,0.0000
C00614=-42.854,-33.363,78.888,155.1350,19.3498,0.0000
C00615=-46.514,-35.238,81.229,154.4158,17.2150,0.0000
C00616=-51.604,-39.197,84.354,153.7972,13.8220,0.0000
C00617=-58.003,-44.233,87.405,158.7585,1.9180,0.0000
C00618=-64.795,-49.536,89.614,-177.4986,1.7097,0.0000
C00619=-70.986,-54.108,90.663,-176.0418,2.8166,0.0000
C00620=-77.451,-55.455,91.206,-175.3401,3.3356,0.0000
C00621=-83.412,-53.310,91.642,-174.9446,3.6075,0.0000
C00622=-87.648,-48.140,92.077,-174.8756,3.6491,0.0000
C00623=-90.907,-41.664,92.362,-174.9695,3.5787,0.0000
C00624=-93.742,-34.820,92.362,173.9131,-1.0168,0.0000
C00625=-96.017,-27.936,92.077,173.7970,-1.0328,0.0000
C00626=-96.677,-21.285,91.642,173.8752,-1.0139,0.0000
C00627=-93.978,-15.553,91.206,174.3470,-0.9286,0.0000
C00628=-88.455,-11.935,90.663,175.2098,-0.8024,0.0000
C00629=-80.844,-10.790,89.614,177.0224,-0.5586,0.0000
C00630=-72.291,-9.737,87.405,-165.9933,16.2421,0.0000
C00631=-64.206,-8.774,84.354,-171.2402,28.1714,0.0000
C00632=-57.808,-7.974,81.229,-174.5367,30.0628,0.0000
C00633=-53.894,-6.711,78.888,-176.9085,30.9855,0.0000
C00634=-52.747,-3.730,77.945,179.1822,31.7634,0.0000
C00635=-52.759,-1.476,77.904,178.6884,31.8401,0.0000
C00636=-52.771,0.000,77.932,179.9987,31.8554,0.0000
C00637=-52.759,1.476,77.904,-178.6868,31.8401,0.0000
C00638=-52.747,3.730,77.945,-179.1836,31.7633,0.0000
C00639=-53.894,6.711,78.888,176.9080,30.9854,0.0000
C00640=-57.808,7.974,81.229,174.5367,30.0629,0.0000
C00641=-64.206,8.774,84.354,171.2403,28.1716,0.0000
C00642=-72.291,9.737,87.405,165.9932,16.2427,0.0000
C00643=-80.844,10.790,89.614,-177.0224,-0.5586,0.0000
C00644=-88.455,11.935,90.663,-175.2098,-0.8024,0.0000
C00645=-93.978,15.553,91.206,-174.3470,-0.9286,0.0000
C00646=-96.677,21.285,91.642,-173.8752,-1.0139,0.0000
C00647=-96.017,27.936,92.077,-173.7970,-1.0328,0.0000
C00648=-93.742,34.820,92.362,-173.9131,-1.0168,0.0000
C00649=-90.907,41.664,92.362,174.9695,3.5787,0.0000
C00650=-87.648,48.140,92.077,174.8756,3.6491,0.0000
C00651=-83.412,53.310,91.642,174.9446,3.6075,0.0000
C00652=-77.451,55.455,91.206,175.3401,3.3356,0.0000
C00653=-70.986,54.108,90.663,176.0418,2.8166,0.0000
C00654=-64.795,49.536,89.614,177.4986,1.7097,0.0000
C00655=-58.003,44.233,87.405,-158.7589,1.9176,0.0000
C00656=-51.604,39.197,84.354,-153.7973,13.8218,0.0000
C00657=-46.514,35.238,81.229,-154.4159,17.2150,0.0000
C00658=-42.854,33.363,78.888,-155.1352,19.3501,0.0000
C00659=-39.935,34.660,77.945,-156.8411,22.3839,0.0000
C00660=-38.350,36.262,77.904,-157.0699,22.7546,0.0000
C00661=-37.314,37.314,77.932,-156.2814,21.9136,0.0000
C00662=-36.262,38.350,77.904,-155.5138,21.0553,0.0000
C00663=-34.660,39.935,77.945,-155.8715,21.3254,0.0000
C00664=-33.363,42.854,78.888,-158.8410,23.3739,0.0000
C00665=-35.238,46.514,81.229,-161.0413,24.3614,0.0000
C00666=-39.197,51.604,84.354,-164.6659,25.3892,0.0000
C00667=-44.233,58.003,87.405,-177.9423,21.2290,0.0000
C00668=-49.536,64.795,89.614,-178.2887,-2.5002,0.0000
C00669=-54.108,70.986,90.663,-177.1767,-3.9534,0.0000
C00670=-55.455,77.451,91.206,-176.6534,-4.6520,0.0000
C00671=-53.310,83.412,91.642,-176.3785,-5.0454,0.0000
C00672=-48.140,87.648,92.077,-176.3363,-5.1140,0.0000
C00673=-41.664,90.907,92.362,-176.4075,-5.0207,0.0000
C00674=-34.820,93.742,92.362,178.9774,6.0859,0.0000
C00675=-27.936,96.017,92.077,178.9611,6.2020,0.0000
C00676=-21.285,96.677,91.642,178.9803,6.1239,0.0000
C00677=-15.553,93.978,91.206,179.0669,5.6522,0.0000
C00678=-11.935,88.455,90.663,179.1947,4.7897,0.0000
C00679=-10.790,80.844,89.614,179.4406,2.9775,0.0000
C00680=-9.737,72.291,87.405,-163.2869,-13.4370,0.0000
C00681=-8.774,64.206,84.354,-151.5477,-7.7153,0.0000
C00682=-7.974,57.808,81.229,-149.8239,-4.7266,0.0000
C00683=-6.711,53.894,78.888,-148.9777,-2.6504,0.0000
C00684=-3.730,52.747,77.945,-148.2341,0.6941,0.0000
C00685=-1.476,52.759,77.904,-148.1532,1.1155,0.0000
C00686=0.000,52.771,77.932,-148.1446,-0.0011,0.0000
C00687=0.000,51.832,79.921,-149.0558,-0.0011,0.0000
C00688=1.391,51.822,79.893,-149.0625,-1.0445,0.0000
C00689=3.586,51.820,79.935,-149.1408,-0.6661,0.0000
C00690=6.543,53.038,80.908,-149.8886,2.6254,0.0000
C00691=7.793,57.125,83.313,-150.7740,4.7141,0.0000
C00692=8.610,63.749,86.500,-152.7472,7.8977,0.0000
C00693=9.608,72.041,89.587,-168.2946,12.4009,0.0000
C00694=10.692,80.728,91.809,179.4187,-3.2869,0.0000
C00695=11.850,88.408,92.861,179.2285,-4.7588,0.0000
C00696=15.484,93.970,93.405,179.1177,-5.5124,0.0000
C00697=21.237,96.685,93.841,179.0403,-5.9433,0.0000
C00698=27.910,96.026,94.277,179.0229,-6.0191,0.0000
C00699=34.811,93.745,94.562,179.0365,-5.9211,0.0000
C00700=41.672,90.903,94.562,-176.4834,4.8629,0.0000
C00701=48.166,87.636,94.277,-176.4231,4.9415,0.0000
C00702=53.350,83.383,93.841,-176.4649,4.8759,0.0000
C00703=55.498,77.395,93.405,-176.7172,4.5175,0.0000
C00704=54.135,70.893,92.861,-177.1748,3.9078,0.0000
C00705=49.523,64.644,91.809,-178.0849,2.7343,0.0000
C00706=44.146,57.735,89.587,179.2966,-16.9755,0.0000
C00707=38.990,51.166,86.500,-165.7542,-24.7012,0.0000
C00708=34.883,45.903,83.313,-161.7994,-23.7154,0.0000
C00709=32.877,42.130,80.908,-159.5645,-22.7531,0.0000
C00710=34.107,39.178,79.935,-156.6314,-20.7599,0.0000
C00711=35.661,37.627,79.893,-156.3055,-20.5225,0.0000
C00712=36.651,36.651,79.921,-157.0254,-21.3204,0.0000
C00713=37.627,35.661,79.893,-157.7666,-22.1091,0.0000
C00714=39.178,34.107,79.935,-157.5618,-21.7697,0.0000
C00715=42.130,32.877,80.908,-155.8881,-18.7825,0.0000
C00716=45.903,34.883,83.313,-155.1829,-16.6167,0.0000
C00717=51.166,38.990,86.500,-154.6124,-12.9186,0.0000
C00718=57.735,44.146,89.587,-163.0228,0.6725,0.0000
C00719=64.644,49.523,91.809,177.2641,-1.9129,0.0000
C00720=70.893,54.135,92.861,176.0875,-2.8186,0.0000
C00721=77.395,55.498,93.405,175.4751,-3.2726,0.0000
C00722=83.383,53.350,93.841,175.1149,-3.5223,0.0000
C00723=87.636,48.166,94.277,175.0489,-3.5635,0.0000
C00724=90.903,41.672,94.562,175.1280,-3.5039,0.0000
C00725=93.745,34.811,94.562,-174.0781,0.9584,0.0000
C00726=96.026,27.910,94.277,-173.9800,0.9717,0.0000
C00727=96.685,21.237,93.841,-174.0558,0.9545,0.0000
C00728=93.970,15.484,93.405,-174.4870,0.8782,0.0000
C00729=88.408,11.850,92.861,-175.2407,0.7688,0.0000
C00730=80.728,10.692,91.809,-176.7129,0.5804,0.0000
C00731=72.041,9.608,89.587,167.3441,-11.4285,0.0000
C00732=63.749,8.610,86.500,171.1309,-26.9732,0.0000
C00733=57.125,7.793,83.313,174.6021,-29.1176,0.0000
C00734=53.038,6.543,80.908,176.9657,-30.0765,0.0000
C00735=51.820,3.586,79.935,-179.2241,-30.8569,0.0000
C00736=51.822,1.391,79.893,-178.7822,-30.9318,0.0000
C00737=51.832,0.000,79.921,-179.9988,-30.9442,0.0000
C00738=51.822,-1.390,79.893,178.7807,-30.9318,0.0000
C00739=51.820,-3.586,79.935,179.2254,-30.8569,0.0000
C00740=53.038,-6.543,80.908,-176.9653,-30.0765,0.0000
C00741=57.125,-7.793,83.313,-174.6020,-29.1177,0.0000
C00742=63.749,-8.610,86.500,-171.1310,-26.9734,0.0000
C00743=72.041,-9.608,89.587,-167.3439,-11.4291,0.0000
C00744=80.728,-10.692,91.809,176.7129,0.5804,0.0000
C00745=88.408,-11.850,92.861,175.2407,0.7688,0.0000
C00746=93.970,-15.484,93.405,174.4870,0.8782,0.0000
C00747=96.685,-21.237,93.841,174.0558,0.9545,0.0000
C00748=96.026,-27.910,94.277,173.9800,0.9717,0.0000
C00749=93.745,-34.811,94.562,174.0781,0.9584,0.0000
C00750=90.903,-41.672,94.562,-175.1280,-3.5039,0.0000
C00751=87.636,-48.166,94.277,-175.0489,-3.5635,0.0000
C00752=83.383,-53.350,93.841,-175.1149,-3.5223,0.0000
C00753=77.395,-55.498,93.405,-175.4751,-3.2726,0.0000
C00754=70.893,-54.135,92.861,-176.0875,-2.8186,0.0000
C00755=64.644,-49.523,91.809,-177.2641,-1.9129,0.0000
C00756=57.735,-44.146,89.587,163.0233,0.6728,0.0000
C00757=51.166,-38.990,86.500,154.6125,-12.9185,0.0000
C00758=45.903,-34.883,83.313,155.1830,-16.6167,0.0000
C00759=42.130,-32.877,80.908,155.8883,-18.7828,0.0000
C00760=39.178,-34.107,79.935,157.5626,-21.7707,0.0000
C00761=37.627,-35.661,79.893,157.7656,-22.1081,0.0000
C00762=36.651,-36.651,79.921,157.0269,-21.3220,0.0000
C00763=35.661,-37.627,79.893,156.3046,-20.5215,0.0000
C00764=34.107,-39.178,79.935,156.6323,-20.7607,0.0000
C00765=32.877,-42.130,80.908,159.5648,-22.7533,0.0000
C00766=34.883,-45.903,83.313,161.7994,-23.7155,0.0000
C00767=38.990,-51.166,86.500,165.7541,-24.7013,0.0000
C00768=44.146,-57.735,89.587,-179.2969,-16.9760,0.0000
C00769=49.523,-64.644,91.809,178.0849,2.7343,0.0000
C00770=54.135,-70.893,92.861,177.1748,3.9078,0.0000
C00771=55.498,-77.395,93.405,176.7172,4.5175,0.0000
C00772=53.350,-83.383,93.841,176.4649,4.8759,0.0000
C00773=48.166,-87.636,94.277,176.4231,4.9415,0.0000
C00774=41.672,-90.903,94.562,176.4834,4.8629,0.0000
C00775=34.811,-93.745,94.562,-179.0365,-5.9211,0.0000
C00776=27.910,-96.026,94.277,-179.0229,-6.0191,0.0000
C00777=21.237,-96.685,93.841,-179.0403,-5.9433,0.0000
C00778=15.484,-93.970,93.405,-179.1177,-5.5124,0.0000
C00779=11.850,-88.408,92.861,-179.2285,-4.7588,0.0000
C00780=10.692,-80.728,91.809,-179.4187,-3.2869,0.0000
C00781=9.608,-72.041,89.587,168.2946,12.4009,0.0000
C00782=8.610,-63.749,86.500,152.7472,7.8977,0.0000
C00783=7.793,-57.125,83.313,150.7740,4.7141,0.0000
C00784=6.543,-53.038,80.908,149.8886,2.6254,0.0000
C00785=3.586,-51.820,79.935,149.1408,-0.6661,0.0000
C00786=1.391,-51.822,79.893,149.0625,-1.0445,0.0000
C00787=0.000,-51.832,79.921,149.0558,-0.0011,0.0000
C00788=0.000,-51.832,79.921,149.0558,-0.0011,0.0000
C00789=-1.390,-51.822,79.893,149.0625,1.0459,0.0000
C00790=-3.586,-51.820,79.935,149.1408,0.6649,0.0000
C00791=-6.543,-53.038,80.908,149.8886,-2.6258,0.0000
C00792=-7.793,-57.125,83.313,150.7739,-4.7142,0.0000
C00793=-8.610,-63.749,86.500,152.7470,-7.8977,0.0000
C00794=-9.608,-72.041,89.587,168.2941,-12.4011,0.0000
C00795=-10.692,-80.728,91.809,-179.4187,3.2869,0.0000
C00796=-11.850,-88.408,92.861,-179.2285,4.7588,0.0000
C00797=-15.484,-93.970,93.405,-179.1177,5.5124,0.0000
C00798=-21.237,-96.685,93.841,-179.0403,5.9433,0.0000
C00799=-27.910,-96.026,94.277,-179.0229,6.0191,0.0000
C00800=-34.811,-93.745,94.562,-179.0365,5.9211,0.0000
C00801=-41.672,-90.903,94.562,176.4834,-4.8629,0.0000
C00802=-48.166,-87.636,94.277,176.4231,-4.9415,0.0000
C00803=-53.350,-83.383,93.841,176.4649,-4.8759,0.0000
C00804=-55.498,-77.395,93.405,176.7172,-4.5175,0.0000
C00805=-54.135,-70.893,92.861,177.1748,-3.9078,0.0000
C00806=-49.523,-64.644,91.809,178.0849,-2.7343,0.0000
C00807=-44.146,-57.735,89.587,-179.2966,16.9755,0.0000
C00808=-38.990,-51.166,86.500,165.7542,24.7012,0.0000
C00809=-34.883,-45.903,83.313,161.7994,23.7154,0.0000
C00810=-32.877,-42.130,80.908,159.5645,22.7531,0.0000
C00811=-34.107,-39.178,79.935,156.6314,20.7599,0.0000
C00812=-35.661,-37.627,79.893,156.3055,20.5225,0.0000
C00813=-36.651,-36.651,79.921,157.0254,21.3204,0.0000
C00814=-37.627,-35.661,79.893,157.7666,22.1091,0.0000
C00815=-39.178,-34.107,79.935,157.5618,21.7697,0.0000
C00816=-42.130,-32.877,80.908,155.8881,18.7825,0.0000
C00817=-45.903,-34.883,83.313,155.1829,16.6167,0.0000
C00818=-51.166,-38.990,86.500,154.6124,12.9186,0.0000
C00819=-57.735,-44.146,89.587,163.0228,-0.6725,0.0000
C00820=-64.644,-49.523,91.809,-177.2641,1.9129,0.0000
C00821=-70.893,-54.135,92.861,-176.0875,2.8186,0.0000
C00822=-77.395,-55.498,93.405,-175.4751,3.2726,0.0000
C00823=-83.383,-53.350,93.841,-175.1149,3.5223,0.0000
C00824=-87.636,-48.166,94.277,-175.0489,3.5635,0.0000
C00825=-90.903,-41.672,94.562,-175.1280,3.5039,0.0000
C00826=-93.745,-34.811,94.562,174.0781,-0.9584,0.0000
C00827=-96.026,-27.910,94.277,173.9800,-0.9717,0.0000
C00828=-96.685,-21.237,93.841,174.0558,-0.9545,0.0000
C00829=-93.970,-15.484,93.405,174.4870,-0.8782,0.0000
C00830=-88.408,-11.850,92.861,175.2407,-0.7688,0.0000
C00831=-80.728,-10.692,91.809,176.7129,-0.5804,0.0000
C00832=-72.041,-9.608,89.587,-167.3441,11.4285,0.0000
C00833=-63.749,-8.610,86.500,-171.1309,26.9732,0.0000
C00834=-57.125,-7.793,83.313,-174.6021,29.1176,0.0000
C00835=-53.038,-6.543,80.908,-176.9657,30.0765,0.0000
C00836=-51.820,-3.586,79.935,179.2241,30.8569,0.0000
C00837=-51.822,-1.391,79.893,178.7822,30.9318,0.0000
C00838=-51.832,0.000,79.921,179.9988,30.9442,0.0000
C00839=-51.822,1.390,79.893,-178.7807,30.9318,0.0000
C00840=-51.820,3.586,79.935,-179.2254,30.8569,0.0000
C00841=-53.038,6.543,80.908,176.9653,30.0765,0.0000
C00842=-57.125,7.793,83.313,174.6020,29.1177,0.0000
C00843=-63.749,8.610,86.500,171.1310,26.9734,0.0000
C00844=-72.041,9.608,89.587,167.3439,11.4291,0.0000
C00845=-80.728,10.692,91.809,-176.7129,-0.5804,0.0000
C00846=-88.408,11.850,92.861,-175.2407,-0.7688,0.0000
C00847=-93.970,15.484,93.405,-174.4870,-0.8782,0.0000
C00848=-96.685,21.237,93.841,-174.0558,-0.9545,0.0000
C00849=-96.026,27.910,94.277,-173.9800,-0.9717,0.0000
C00850=-93.745,34.811,94.562,-174.0781,-0.9584,0.0000
C00851=-90.903,41.672,94.562,175.1280,3.5039,0.0000
C00852=-87.636,48.166,94.277,175.0489,3.5635,0.0000
C00853=-83.383,53.350,93.841,175.1149,3.5223,0.0000
C00854=-77.395,55.498,93.405,175.4751,3.2726,0.0000
C00855=-70.893,54.135,92.861,176.0875,2.8186,0.0000
C00856=-64.644,49.523,91.809,177.2641,1.9129,0.0000
C00857=-57.735,44.146,89.587,-163.0233,-0.6728,0.0000
C00858=-51.166,38.990,86.500,-154.6125,12.9185,0.0000
C00859=-45.903,34.883,83.313,-155.1830,16.6167,0.0000
C00860=-42.130,32.877,80.908,-155.8883,18.7828,0.0000
C00861=-39.178,34.107,79.935,-157.5626,21.7707,0.0000
C00862=-37.627,35.661,79.893,-157.7656,22.1081,0.0000
C00863=-36.651,36.651,79.921,-157.0269,21.3220,0.0000
C00864=-35.661,37.627,79.893,-156.3046,20.5215,0.0000
C00865=-34.107,39.178,79.935,-156.6323,20.7607,0.0000
C00866=-32.877,42.130,80.908,-159.5648,22.7533,0.0000
C00867=-34.883,45.903,83.313,-161.7994,23.7155,0.0000
C00868=-38.990,51.166,86.500,-165.7541,24.7013,0.0000
C00869=-44.146,57.735,89.587,179.2969,16.9760,0.0000
C00870=-49.523,64.644,91.809,-178.0849,-2.7343,0.0000
C00871=-54.135,70.893,92.861,-177.1748,-3.9078,0.0000
C00872=-55.498,77.395,93.405,-176.7172,-4.5175,0.0000
C00873=-53.350,83.383,93.841,-176.4649,-4.8759,0.0000
C00874=-48.166,87.636,94.277,-176.4231,-4.9415,0.0000
C00875=-41.672,90.903,94.562,-176.4834,-4.8629,0.0000
C00876=-34.811,93.745,94.562,179.0365,5.9211,0.0000
C00877=-27.910,96.026,94.277,179.0229,6.0191,0.0000
C00878=-21.237,96.685,93.841,179.0403,5.9433,0.0000
C00879=-15.484,93.970,93.405,179.1177,5.5124,0.0000
C00880=-11.850,88.408,92.861,179.2285,4.7588,0.0000
C00881=-10.692,80.728,91.809,179.4187,3.2869,0.0000
C00882=-9.608,72.041,89.587,-168.2941,-12.4011,0.0000
C00883=-8.610,63.749,86.500,-152.7470,-7.8977,0.0000
C00884=-7.793,57.125,83.313,-150.7739,-4.7142,0.0000
C00885=-6.543,53.038,80.908,-149.8886,-2.6258,0.0000
C00886=-3.586,51.820,79.935,-149.1408,0.6649,0.0000
C00887=-1.390,51.822,79.893,-149.0625,1.0459,0.0000
C00888=0.000,51.832,79.921,-149.0558,-0.0011,0.0000
C00889=0.000,50.970,81.946,-150.0295,-0.0010,0.0000
C00890=1.312,50.962,81.916,-150.0342,-0.9747,0.0000
C00891=3.453,50.970,81.960,-150.1104,-0.6322,0.0000
C00892=6.389,52.261,82.960,-150.8663,2.6038,0.0000
C00893=7.633,56.525,85.423,-151.8048,4.7130,0.0000
C00894=8.475,63.374,88.663,-154.1050,8.1144,0.0000
C00895=9.515,71.858,91.777,-174.1964,9.1640,0.0000
C00896=10.634,80.658,94.007,179.4190,-3.4601,0.0000
C00897=11.808,88.386,95.061,179.2691,-4.6583,0.0000
C00898=15.455,93.966,95.604,179.1732,-5.3156,0.0000
C00899=55.516,77.372,95.604,-176.8180,4.3396,0.0000
C00900=54.149,70.847,95.061,-177.2176,3.8082,0.0000
C00901=49.515,64.553,94.007,-177.9619,2.8565,0.0000
C00902=44.083,57.539,91.777,177.5499,-10.5564,0.0000
C00903=38.820,50.805,88.663,-166.9816,-23.9241,0.0000
C00904=34.571,45.367,85.423,-162.6237,-23.0206,0.0000
C00905=32.436,41.472,82.960,-160.3381,-22.0875,0.0000
C00906=33.599,38.483,81.960,-157.4403,-20.1543,0.0000
C00907=35.108,36.963,81.916,-157.1411,-19.9444,0.0000
C00908=36.041,36.041,81.946,-157.8154,-20.6847,0.0000
C00909=36.963,35.108,81.916,-158.5065,-21.4187,0.0000
C00910=38.483,33.599,81.960,-158.3247,-21.1088,0.0000
C00911=41.472,32.436,82.960,-156.6871,-18.1660,0.0000
C00912=45.367,34.571,85.423,-156.0005,-15.9539,0.0000
C00913=50.805,38.820,88.663,-155.5180,-11.8829,0.0000
C00914=57.539,44.083,91.777,-169.4338,2.4086,0.0000
C00915=64.553,49.515,94.007,177.1417,-2.0355,0.0000
C00916=70.847,54.149,95.061,176.1874,-2.7763,0.0000
C00917=77.372,55.516,95.604,175.6538,-3.1729,0.0000
C00918=93.966,15.455,95.604,-174.6838,0.8232,0.0000
C00919=88.386,11.808,95.061,-175.3413,0.7285,0.0000
C00920=80.658,10.634,94.007,-176.5397,0.5800,0.0000
C00921=71.858,9.515,91.777,170.7896,-5.7292,0.0000
C00922=63.374,8.475,88.663,170.9941,-25.6168,0.0000
C00923=56.525,7.633,85.423,174.6559,-28.0914,0.0000
C00924=52.261,6.389,82.960,177.0197,-29.1007,0.0000
C00925=50.970,3.453,81.960,-179.2708,-29.8876,0.0000
C00926=50.962,1.312,81.916,-178.8749,-29.9610,0.0000
C00927=50.970,0.000,81.946,-179.9988,-29.9705,0.0000
C00928=50.962,-1.311,81.916,178.8734,-29.9610,0.0000
C00929=50.970,-3.454,81.960,179.2721,-29.8876,0.0000
C00930=52.261,-6.389,82.960,-177.0193,-29.1007,0.0000
C00931=56.525,-7.633,85.423,-174.6559,-28.0915,0.0000
C00932=63.374,-8.475,88.663,-170.9942,-25.6170,0.0000
C00933=71.858,-9.515,91.777,-170.7893,-5.7295,0.0000
C00934=80.658,-10.634,94.007,176.5397,0.5800,0.0000
C00935=88.386,-11.808,95.061,175.3413,0.7285,0.0000
C00936=93.966,-15.455,95.604,174.6838,0.8232,0.0000
C00937=77.372,-55.516,95.604,-175.6538,-3.1729,0.0000
C00938=70.847,-54.149,95.061,-176.1874,-2.7763,0.0000
C00939=64.553,-49.515,94.007,-177.1417,-2.0355,0.0000
C00940=57.539,-44.083,91.777,169.4341,2.4086,0.0000
C00941=50.805,-38.820,88.663,155.5181,-11.8828,0.0000
C00942=45.367,-34.571,85.423,156.0006,-15.9539,0.0000
C00943=41.472,-32.436,82.960,156.6873,-18.1663,0.0000
C00944=38.483,-33.599,81.960,158.3254,-21.1097,0.0000
C00945=36.963,-35.108,81.916,158.5056,-21.4177,0.0000
C00946=36.041,-36.041,81.946,157.8169,-20.6863,0.0000
C00947=35.108,-36.963,81.916,157.1402,-19.9433,0.0000
C00948=33.599,-38.483,81.960,157.4412,-20.1551,0.0000
C00949=32.436,-41.472,82.960,160.3384,-22.0878,0.0000
C00950=34.571,-45.367,85.423,162.6237,-23.0206,0.0000
C00951=38.820,-50.805,88.663,166.9814,-23.9241,0.0000
C00952=44.083,-57.539,91.777,-177.5499,-10.5568,0.0000
C00953=49.515,-64.553,94.007,177.9619,2.8565,0.0000
C00954=54.149,-70.847,95.061,177.2176,3.8082,0.0000
C00955=55.516,-77.372,95.604,176.8180,4.3396,0.0000
C00956=15.455,-93.966,95.604,-179.1732,-5.3156,0.0000
C00957=11.808,-88.386,95.061,-179.2691,-4.6583,0.0000
C00958=10.634,-80.658,94.007,-179.4190,-3.4601,0.0000
C00959=9.515,-71.858,91.777,174.1964,9.1640,0.0000
C00960=8.475,-63.374,88.663,154.1050,8.1144,0.0000
C00961=7.633,-56.525,85.423,151.8048,4.7130,0.0000
C00962=6.389,-52.261,82.960,150.8663,2.6038,0.0000
C00963=3.453,-50.970,81.960,150.1104,-0.6322,0.0000
C00964=1.312,-50.962,81.916,150.0342,-0.9747,0.0000
C00965=0.000,-50.970,81.946,150.0295,-0.0010,0.0000
C00966=0.000,-50.970,81.946,150.0295,-0.0010,0.0000
C00967=-1.311,-50.962,81.916,150.0342,0.9761,0.0000
C00968=-3.454,-50.970,81.960,150.1104,0.6311,0.0000
C00969=-6.389,-52.261,82.960,150.8663,-2.6042,0.0000
C00970=-7.633,-56.525,85.423,151.8047,-4.7130,0.0000
C00971=-8.475,-63.374,88.663,154.1049,-8.1143,0.0000
C00972=-9.515,-71.858,91.777,174.1961,-9.1643,0.0000
C00973=-10.634,-80.658,94.007,-179.4190,3.4601,0.0000
C00974=-11.808,-88.386,95.061,-179.2691,4.6583,0.0000
C00975=-15.455,-93.966,95.604,-179.1732,5.3156,0.0000
C00976=-55.516,-77.372,95.604,176.8180,-4.3396,0.0000
C00977=-54.149,-70.847,95.061,177.2176,-3.8082,0.0000
C00978=-49.515,-64.553,94.007,177.9619,-2.8565,0.0000
C00979=-44.083,-57.539,91.777,-177.5499,10.5564,0.0000
C00980=-38.820,-50.805,88.663,166.9816,23.9241,0.0000
C00981=-34.571,-45.367,85.423,162.6237,23.0206,0.0000
C00982=-32.436,-41.472,82.960,160.3381,22.0875,0.0000
C00983=-33.599,-38.483,81.960,157.4403,20.1543,0.0000
C00984=-35.108,-36.963,81.916,157.1411,19.9444,0.0000
C00985=-36.041,-36.041,81.946,157.8154,20.6847,0.0000
C00986=-36.963,-35.108,81.916,158.5065,21.4187,0.0000
C00987=-38.483,-33.599,81.960,158.3247,21.1088,0.0000
C00988=-41.472,-32.436,82.960,156.6871,18.1660,0.0000
C00989=-45.367,-34.571,85.423,156.0005,15.9539,0.0000
C00990=-50.805,-38.820,88.663,155.5180,11.8829,0.0000
C00991=-57.539,-44.083,91.777,169.4338,-2.4086,0.0000
C00992=-64.553,-49.515,94.007,-177.1417,2.0355,0.0000
C00993=-70.847,-54.149,95.061,-176.1874,2.7763,0.0000
C00994=-77.372,-55.516,95.604,-175.6538,3.1729,0.0000
C00995=-93.966,-15.455,95.604,174.6838,-0.8232,0.0000
C00996=-88.386,-11.808,95.061,175.3413,-0.7285,0.0000
C00997=-80.658,-10.634,94.007,176.5397,-0.5800,0.0000
C00998=-71.858,-9.515,91.777,-170.7896,5.7292,0.0000
C00999=-63.374,-8.475,88.663,-170.9941,25.6168,0.0000
C01000=-56.525,-7.633,85.423,-174.6559,28.0914,0.0000
C01001=-52.261,-6.389,82.960,-177.0197,29.1007,0.0000
C01002=-50.970,-3.453,81.960,179.2708,29.8876,0.0000
C01003=-50.962,-1.312,81.916,178.8749,29.9610,0.0000
C01004=-50.970,0.000,81.946,179.9988,29.9705,0.0000
C01005=-50.962,1.311,81.916,-178.8734,29.9610,0.0000
C01006=-50.970,3.454,81.960,-179.2721,29.8876,0.0000
C01007=-52.261,6.389,82.960,177.0193,29.1007,0.0000
C01008=-56.525,7.633,85.423,174.6559,28.0915,0.0000
C01009=-63.374,8.475,88.663,170.9942,25.6170,0.0000
C01010=-71.858,9.515,91.777,170.7893,5.7295,0.0000
C01011=-80.658,10.634,94.007,-176.5397,-0.5800,0.0000
C01012=-88.386,11.808,95.061,-175.3413,-0.7285,0.0000
C01013=-93.966,15.455,95.604,-174.6838,-0.8232,0.0000
C01014=-77.372,55.516,95.604,175.6538,3.1729,0.0000
C01015=-70.847,54.149,95.061,176.1874,2.7763,0.0000
C01016=-64.553,49.515,94.007,177.1417,2.0355,0.0000
C01017=-57.539,44.083,91.777,-169.4341,-2.4086,0.0000
C01018=-50.805,38.820,88.663,-155.5181,11.8828,0.0000
C01019=-45.367,34.571,85.423,-156.0006,15.9539,0.0000
C01020=-41.472,32.436,82.960,-156.6873,18.1663,0.0000
C01021=-38.483,33.599,81.960,-158.3254,21.1097,0.0000
C01022=-36.963,35.108,81.916,-158.5056,21.4177,0.0000
C01023=-36.041,36.041,81.946,-157.8169,20.6863,0.0000
C01024=-35.108,36.963,81.916,-157.1402,19.9433,0.0000
C01025=-33.599,38.483,81.960,-157.4412,20.1551,0.0000
C01026=-32.436,41.472,82.960,-160.3384,22.0878,0.0000
C01027=-34.571,45.367,85.423,-162.6237,23.0206,0.0000
C01028=-38.820,50.805,88.663,-166.9814,23.9241,0.0000
C01029=-44.083,57.539,91.777,177.5499,10.5568,0.0000
C01030=-49.515,64.553,94.007,-177.9619,-2.8565,0.0000
C01031=-54.149,70.847,95.061,-177.2176,-3.8082,0.0000
C01032=-55.516,77.372,95.604,-176.8180,-4.3396,0.0000
C01033=-15.455,93.966,95.604,179.1732,5.3156,0.0000
C01034=-11.808,88.386,95.061,179.2691,4.6583,0.0000
C01035=-10.634,80.658,94.007,179.4190,3.4601,0.0000
C01036=-9.515,71.858,91.777,-174.1961,-9.1643,0.0000
C01037=-8.475,63.374,88.663,-154.1049,-8.1143,0.0000
C01038=-7.633,56.525,85.423,-151.8047,-4.7130,0.0000
C01039=-6.389,52.261,82.960,-150.8663,-2.6042,0.0000
C01040=-3.454,50.970,81.960,-150.1104,0.6311,0.0000
C01041=-1.311,50.962,81.916,-150.0342,0.9761,0.0000
C01042=0.000,50.970,81.946,-150.0295,-0.0010,0.0000
C01043=0.000,50.195,84.004,-151.0670,-0.0010,0.0000
C01044=1.241,50.188,83.974,-151.0698,-0.9055,0.0000
C01045=3.334,50.204,84.019,-151.1443,-0.5925,0.0000
C01046=6.253,51.571,85.045,-151.9132,2.5872,0.0000
C01047=7.499,56.017,87.559,-152.9216,4.7257,0.0000
C01048=8.371,63.087,90.842,-155.6526,8.3629,0.0000
C01049=9.459,71.748,93.974,-179.0563,2.8494,0.0000
C01050=44.045,57.421,93.974,178.6508,-2.6814,0.0000
C01051=38.690,50.529,90.842,-168.3665,-23.0330,0.0000
C01052=34.307,44.912,87.559,-163.5188,-22.2744,0.0000
C01053=32.045,40.888,85.045,-161.1637,-21.3763,0.0000
C01054=33.142,37.857,84.019,-158.2984,-19.5071,0.0000
C01055=34.611,36.365,83.974,-158.0210,-19.3198,0.0000
C01056=35.493,35.493,84.004,-158.6500,-20.0034,0.0000
C01057=36.365,34.611,83.974,-159.2913,-20.6835,0.0000
C01058=37.858,33.142,84.019,-159.1283,-20.3976,0.0000
C01059=40.888,32.045,85.045,-157.5314,-17.4966,0.0000
C01060=44.912,34.307,87.559,-156.8697,-15.2204,0.0000
C01061=50.529,38.690,90.842,-156.5355,-10.6948,0.0000
C01062=57.421,44.045,93.974,-177.3178,1.3477,0.0000
C01063=71.748,9.459,93.974,177.1503,-0.9425,0.0000
C01064=63.087,8.371,90.842,170.8339,-24.0720,0.0000
C01065=56.017,7.499,87.559,174.6956,-26.9789,0.0000
C01066=51.571,6.253,85.045,177.0680,-28.0556,0.0000
C01067=50.204,3.334,84.019,-179.3235,-28.8540,0.0000
C01068=50.188,1.241,83.974,-178.9654,-28.9262,0.0000
C01069=50.195,0.000,84.004,-179.9989,-28.9330,0.0000
C01070=50.188,-1.240,83.974,178.9640,-28.9262,0.0000
C01071=50.204,-3.335,84.019,179.3248,-28.8540,0.0000
C01072=51.571,-6.253,85.045,-177.0677,-28.0556,0.0000
C01073=56.017,-7.499,87.559,-174.6956,-26.9789,0.0000
C01074=63.087,-8.371,90.842,-170.8340,-24.0722,0.0000
C01075=71.748,-9.459,93.974,-177.1502,-0.9425,0.0000
C01076=57.421,-44.045,93.974,177.3179,1.3477,0.0000
C01077=50.529,-38.690,90.842,156.5357,-10.6946,0.0000
C01078=44.912,-34.307,87.559,156.8698,-15.2203,0.0000
C01079=40.888,-32.045,85.045,157.5316,-17.4969,0.0000
C01080=37.857,-33.142,84.019,159.1290,-20.3985,0.0000
C01081=36.365,-34.611,83.974,159.2904,-20.6825,0.0000
C01082=35.493,-35.493,84.004,158.6514,-20.0049,0.0000
C01083=34.611,-36.365,83.974,158.0201,-19.3188,0.0000
C01084=33.142,-37.858,84.019,158.2993,-19.5079,0.0000
C01085=32.045,-40.888,85.045,161.1640,-21.3765,0.0000
C01086=34.307,-44.912,87.559,163.5187,-22.2745,0.0000
C01087=38.690,-50.529,90.842,168.3664,-23.0331,0.0000
C01088=44.045,-57.421,93.974,-178.6508,-2.6815,0.0000
C01089=9.459,-71.748,93.974,179.0563,2.8494,0.0000
C01090=8.371,-63.087,90.842,155.6526,8.3629,0.0000
C01091=7.499,-56.017,87.559,152.9216,4.7257,0.0000
C01092=6.253,-51.571,85.045,151.9132,2.5872,0.0000
C01093=3.334,-50.204,84.019,151.1443,-0.5925,0.0000
C01094=1.241,-50.188,83.974,151.0698,-0.9055,0.0000
C01095=0.000,-50.195,84.004,151.0670,-0.0010,0.0000
C01096=0.000,-50.195,84.004,151.0670,-0.0010,0.0000
C01097=-1.240,-50.188,83.974,151.0698,0.9068,0.0000
C01098=-3.335,-50.204,84.019,151.1444,0.5914,0.0000
C01099=-6.253,-51.571,85.045,151.9132,-2.5875,0.0000
C01100=-7.499,-56.017,87.559,152.9215,-4.7258,0.0000
C01101=-8.371,-63.087,90.842,155.6524,-8.3629,0.0000
C01102=-9.459,-71.748,93.974,179.0563,-2.8495,0.0000
C01103=-44.045,-57.421,93.974,-178.6508,2.6814,0.0000
C01104=-38.690,-50.529,90.842,168.3665,23.0330,0.0000
C01105=-34.307,-44.912,87.559,163.5188,22.2744,0.0000
C01106=-32.045,-40.888,85.045,161.1637,21.3763,0.0000
C01107=-33.142,-37.857,84.019,158.2984,19.5071,0.0000
C01108=-34.611,-36.365,83.974,158.0210,19.3198,0.0000
C01109=-35.493,-35.493,84.004,158.6500,20.0034,0.0000
C01110=-36.365,-34.611,83.974,159.2913,20.6835,0.0000
C01111=-37.858,-33.142,84.019,159.1283,20.3976,0.0000
C01112=-40.888,-32.045,85.045,157.5314,17.4966,0.0000
C01113=-44.912,-34.307,87.559,156.8697,15.2204,0.0000
C01114=-50.529,-38.690,90.842,156.5355,10.6948,0.0000
C01115=-57.421,-44.045,93.974,177.3178,-1.3477,0.0000
C01116=-71.748,-9.459,93.974,-177.1503,0.9425,0.0000
C01117=-63.087,-8.371,90.842,-170.8339,24.0720,0.0000
C01118=-56.017,-7.499,87.559,-174.6956,26.9789,0.0000
C01119=-51.571,-6.253,85.045,-177.0680,28.0556,0.0000
C01120=-50.204,-3.334,84.019,179.3235,28.8540,0.0000
C01121=-50.188,-1.241,83.974,178.9654,28.9262,0.0000
C01122=-50.195,0.000,84.004,179.9989,28.9330,0.0000
C01123=-50.188,1.240,83.974,-178.9640,28.9262,0.0000
C01124=-50.204,3.335,84.019,-179.3248,28.8540,0.0000
C01125=-51.571,6.253,85.045,177.0677,28.0556,0.0000
C01126=-56.017,7.499,87.559,174.6956,26.9789,0.0000
C01127=-63.087,8.371,90.842,170.8340,24.0722,0.0000
C01128=-71.748,9.459,93.974,177.1502,0.9425,0.0000
C01129=-57.421,44.045,93.974,-177.3179,-1.3477,0.0000
C01130=-50.529,38.690,90.842,-156.5357,10.6946,0.0000
C01131=-44.912,34.307,87.559,-156.8698,15.2203,0.0000
C01132=-40.888,32.045,85.045,-157.5316,17.4969,0.0000
C01133=-37.857,33.142,84.019,-159.1290,20.3985,0.0000
C01134=-36.365,34.611,83.974,-159.2904,20.6825,0.0000
C01135=-35.493,35.493,84.004,-158.6514,20.0049,0.0000
C01136=-34.611,36.365,83.974,-158.0201,19.3188,0.0000
C01137=-33.142,37.858,84.019,-158.2993,19.5079,0.0000
C01138=-32.045,40.888,85.045,-161.1640,21.3765,0.0000
C01139=-34.307,44.912,87.559,-163.5187,22.2745,0.0000
C01140=-38.690,50.529,90.842,-168.3664,23.0331,0.0000
C01141=-44.045,57.421,93.974,178.6508,2.6815,0.0000
C01142=-9.459,71.748,93.974,-179.0563,-2.8495,0.0000
C01143=-8.371,63.087,90.842,-155.6524,-8.3629,0.0000
C01144=-7.499,56.017,87.559,-152.9215,-4.7258,0.0000
C01145=-6.253,51.571,85.045,-151.9132,-2.5875,0.0000
C01146=-3.335,50.204,84.019,-151.1444,0.5914,0.0000
C01147=-1.240,50.188,83.974,-151.0698,0.9068,0.0000
C01148=0.000,50.195,84.004,-151.0670,-0.0010,0.0000
C01149=0.000,49.517,86.097,-152.1693,-0.0009,0.0000
C01150=1.179,49.510,86.067,-152.1704,-0.8376,0.0000
C01151=3.230,49.536,86.112,-152.2437,-0.5457,0.0000
C01152=6.137,50.981,87.161,-153.0315,2.5775,0.0000
C01153=7.391,55.610,89.719,-154.1304,4.7546,0.0000
C01154=8.302,62.896,93.033,-157.4301,8.6331,0.0000
C01155=38.603,50.345,93.033,-169.9269,-21.9910,0.0000
C01156=34.096,44.548,89.719,-164.4893,-21.4739,0.0000
C01157=31.710,40.389,87.161,-162.0433,-20.6187,0.0000
C01158=32.743,37.311,86.112,-159.2064,-18.8178,0.0000
C01159=34.176,35.843,86.067,-158.9446,-18.6470,0.0000
C01160=35.014,35.014,86.097,-159.5288,-19.2753,0.0000
C01161=35.842,34.176,86.067,-160.1213,-19.9028,0.0000
C01162=37.311,32.743,86.112,-159.9717,-19.6342,0.0000
C01163=40.389,31.710,87.161,-158.4203,-16.7709,0.0000
C01164=44.548,34.096,89.719,-157.7921,-14.4099,0.0000
C01165=50.345,38.603,93.033,-157.6981,-9.3335,0.0000
C01166=62.896,8.302,93.033,170.6630,-22.3003,0.0000
C01167=55.610,7.391,89.719,174.7188,-25.7740,0.0000
C01168=50.981,6.137,87.161,177.1085,-26.9390,0.0000
C01169=49.536,3.230,86.112,-179.3834,-27.7549,0.0000
C01170=49.510,1.179,86.067,-179.0529,-27.8264,0.0000
C01171=49.517,0.000,86.097,-179.9989,-27.8307,0.0000
C01172=49.510,-1.178,86.067,179.0515,-27.8264,0.0000
C01173=49.536,-3.231,86.112,179.3846,-27.7549,0.0000
C01174=50.981,-6.137,87.161,-177.1082,-26.9390,0.0000
C01175=55.610,-7.391,89.719,-174.7187,-25.7741,0.0000
C01176=62.896,-8.302,93.033,-170.6630,-22.3005,0.0000
C01177=50.345,-38.603,93.033,157.6982,-9.3334,0.0000
C01178=44.548,-34.096,89.719,157.7922,-14.4098,0.0000
C01179=40.389,-31.710,87.161,158.4205,-16.7712,0.0000
C01180=37.311,-32.743,86.112,159.9724,-19.6350,0.0000
C01181=35.843,-34.176,86.067,160.1204,-19.9019,0.0000
C01182=35.014,-35.014,86.097,159.5301,-19.2768,0.0000
C01183=34.176,-35.842,86.067,158.9438,-18.6461,0.0000
C01184=32.743,-37.311,86.112,159.2072,-18.8185,0.0000
C01185=31.710,-40.389,87.161,162.0435,-20.6190,0.0000
C01186=34.096,-44.548,89.719,164.4892,-21.4740,0.0000
C01187=38.603,-50.345,93.033,169.9267,-21.9911,0.0000
C01188=8.302,-62.896,93.033,157.4301,8.6331,0.0000
C01189=7.391,-55.610,89.719,154.1304,4.7546,0.0000
C01190=6.137,-50.981,87.161,153.0315,2.5775,0.0000
C01191=3.230,-49.536,86.112,152.2437,-0.5457,0.0000
C01192=1.179,-49.510,86.067,152.1704,-0.8376,0.0000
C01193=0.000,-49.517,86.097,152.1693,-0.0009,0.0000
C01194=0.000,-49.517,86.097,152.1693,-0.0009,0.0000
C01195=-1.178,-49.510,86.067,152.1704,0.8389,0.0000
C01196=-3.231,-49.536,86.112,152.2438,0.5446,0.0000
C01197=-6.137,-50.981,87.161,153.0315,-2.5778,0.0000
C01198=-7.391,-55.610,89.719,154.1303,-4.7546,0.0000
C01199=-8.302,-62.896,93.033,157.4299,-8.6331,0.0000
C01200=-38.603,-50.345,93.033,169.9269,21.9910,0.0000
C01201=-34.096,-44.548,89.719,164.4893,21.4739,0.0000
C01202=-31.710,-40.389,87.161,162.0433,20.6187,0.0000
C01203=-32.743,-37.311,86.112,159.2064,18.8178,0.0000
C01204=-34.176,-35.843,86.067,158.9446,18.6470,0.0000
C01205=-35.014,-35.014,86.097,159.5288,19.2753,0.0000
C01206=-35.842,-34.176,86.067,160.1213,19.9028,0.0000
C01207=-37.311,-32.743,86.112,159.9717,19.6342,0.0000
C01208=-40.389,-31.710,87.161,158.4203,16.7709,0.0000
C01209=-44.548,-34.096,89.719,157.7921,14.4099,0.0000
C01210=-50.345,-38.603,93.033,157.6981,9.3335,0.0000
C01211=-62.896,-8.302,93.033,-170.6630,22.3003,0.0000
C01212=-55.610,-7.391,89.719,-174.7188,25.7740,0.0000
C01213=-50.981,-6.137,87.161,-177.1085,26.9390,0.0000
C01214=-49.536,-3.230,86.112,179.3834,27.7549,0.0000
C01215=-49.510,-1.179,86.067,179.0529,27.8264,0.0000
C01216=-49.517,0.000,86.097,179.9989,27.8307,0.0000
C01217=-49.510,1.178,86.067,-179.0515,27.8264,0.0000
C01218=-49.536,3.231,86.112,-179.3846,27.7549,0.0000
C01219=-50.981,6.137,87.161,177.1082,26.9390,0.0000
C01220=-55.610,7.391,89.719,174.7187,25.7741,0.0000
C01221=-62.896,8.302,93.033,170.6630,22.3005,0.0000
C01222=-50.345,38.603,93.033,-157.6982,9.3334,0.0000
C01223=-44.548,34.096,89.719,-157.7922,14.4098,0.0000
C01224=-40.389,31.710,87.161,-158.4205,16.7712,0.0000
C01225=-37.311,32.743,86.112,-159.9724,19.6350,0.0000
C01226=-35.843,34.176,86.067,-160.1204,19.9019,0.0000
C01227=-35.014,35.014,86.097,-159.5301,19.2768,0.0000
C01228=-34.176,35.842,86.067,-158.9438,18.6461,0.0000
C01229=-32.743,37.311,86.112,-159.2072,18.8185,0.0000
C01230=-31.710,40.389,87.161,-162.0435,20.6190,0.0000
C01231=-34.096,44.548,89.719,-164.4892,21.4740,0.0000
C01232=-38.603,50.345,93.033,-169.9267,21.9911,0.0000
C01233=-8.302,62.896,93.033,-157.4299,-8.6331,0.0000
C01234=-7.391,55.610,89.719,-154.1303,-4.7546,0.0000
C01235=-6.137,50.981,87.161,-153.0315,-2.5778,0.0000
C01236=-3.231,49.536,86.112,-152.2438,0.5446,0.0000
C01237=-1.178,49.510,86.067,-152.1704,0.8389,0.0000
C01238=0.000,49.517,86.097,-152.1693,-0.0009,0.0000
C01239=0.000,48.949,88.223,-153.3370,-0.0009,0.0000
C01240=1.127,48.942,88.191,-153.3363,-0.7719,0.0000
C01241=3.143,48.975,88.238,-153.4093,-0.4906,0.0000
C01242=6.042,50.501,89.306,-154.2231,2.5765,0.0000
C01243=7.312,55.314,91.898,-155.4376,4.8010,0.0000
C01244=8.270,62.805,95.231,-159.4886,8.8986,0.0000
C01245=38.562,50.258,95.231,-171.6749,-20.7421,0.0000
C01246=33.942,44.284,91.898,-165.5397,-20.6148,0.0000
C01247=31.437,39.982,89.306,-162.9784,-19.8144,0.0000
C01248=32.408,36.853,88.238,-160.1646,-18.0861,0.0000
C01249=33.811,35.404,88.191,-159.9107,-17.9244,0.0000
C01250=34.612,34.612,88.223,-160.4512,-18.4996,0.0000
C01251=35.404,33.811,88.191,-160.9963,-19.0763,0.0000
C01252=36.854,32.408,88.238,-160.8535,-18.8166,0.0000
C01253=39.982,31.437,89.306,-159.3528,-15.9857,0.0000
C01254=44.284,33.942,91.898,-158.7699,-13.5163,0.0000
C01255=50.258,38.562,95.231,-159.0559,-7.7821,0.0000
C01256=62.805,8.270,95.231,170.5097,-20.2536,0.0000
C01257=55.314,7.312,91.898,174.7239,-24.4706,0.0000
C01258=50.501,6.042,89.306,177.1393,-25.7489,0.0000
C01259=48.975,3.143,88.238,-179.4514,-26.5896,0.0000
C01260=48.942,1.127,88.191,-179.1363,-26.6610,0.0000
C01261=48.949,0.000,88.223,-179.9990,-26.6630,0.0000
C01262=48.942,-1.126,88.191,179.1350,-26.6610,0.0000
C01263=48.976,-3.143,88.238,179.4525,-26.5896,0.0000
C01264=50.501,-6.042,89.306,-177.1390,-25.7489,0.0000
C01265=55.314,-7.312,91.898,-174.7238,-24.4707,0.0000
C01266=62.805,-8.270,95.231,-170.5097,-20.2538,0.0000
C01267=50.258,-38.562,95.231,159.0560,-7.7820,0.0000
C01268=44.284,-33.942,91.898,158.7700,-13.5162,0.0000
C01269=39.982,-31.437,89.306,159.3530,-15.9859,0.0000
C01270=36.853,-32.408,88.238,160.8541,-18.8174,0.0000
C01271=35.404,-33.811,88.191,160.9955,-19.0754,0.0000
C01272=34.612,-34.612,88.223,160.4524,-18.5009,0.0000
C01273=33.811,-35.404,88.191,159.9099,-17.9235,0.0000
C01274=32.408,-36.854,88.238,160.1654,-18.0867,0.0000
C01275=31.437,-39.982,89.306,162.9786,-19.8146,0.0000
C01276=33.942,-44.284,91.898,165.5396,-20.6149,0.0000
C01277=38.562,-50.258,95.231,171.6748,-20.7423,0.0000
C01278=8.270,-62.805,95.231,159.4886,8.8986,0.0000
C01279=7.312,-55.314,91.898,155.4376,4.8010,0.0000
C01280=6.042,-50.501,89.306,154.2231,2.5765,0.0000
C01281=3.143,-48.975,88.238,153.4093,-0.4906,0.0000
C01282=1.127,-48.942,88.191,153.3363,-0.7719,0.0000
C01283=0.000,-48.949,88.223,153.3370,-0.0009,0.0000
C01284=0.000,-48.949,88.223,153.3370,-0.0009,0.0000
C01285=-1.126,-48.942,88.191,153.3363,0.7730,0.0000
C01286=-3.143,-48.976,88.238,153.4094,0.4896,0.0000
C01287=-6.042,-50.501,89.306,154.2231,-2.5767,0.0000
C01288=-7.312,-55.314,91.898,155.4374,-4.8011,0.0000
C01289=-8.270,-62.805,95.231,159.4884,-8.8986,0.0000
C01290=-38.562,-50.258,95.231,171.6749,20.7421,0.0000
C01291=-33.942,-44.284,91.898,165.5397,20.6148,0.0000
C01292=-31.437,-39.982,89.306,162.9784,19.8144,0.0000
C01293=-32.408,-36.853,88.238,160.1646,18.0861,0.0000
C01294=-33.811,-35.404,88.191,159.9107,17.9244,0.0000
C01295=-34.612,-34.612,88.223,160.4512,18.4996,0.0000
C01296=-35.404,-33.811,88.191,160.9963,19.0763,0.0000
C01297=-36.854,-32.408,88.238,160.8535,18.8166,0.0000
C01298=-39.982,-31.437,89.306,159.3528,15.9857,0.0000
C01299=-44.284,-33.942,91.898,158.7699,13.5163,0.0000
C01300=-50.258,-38.562,95.231,159.0559,7.7821,0.0000
C01301=-62.805,-8.270,95.231,-170.5097,20.2536,0.0000
C01302=-55.314,-7.312,91.898,-174.7239,24.4706,0.0000
C01303=-50.501,-6.042,89.306,-177.1393,25.7489,0.0000
C01304=-48.975,-3.143,88.238,179.4514,26.5896,0.0000
C01305=-48.942,-1.127,88.191,179.1363,26.6610,0.0000
C01306=-48.949,0.000,88.223,179.9990,26.6630,0.0000
C01307=-48.942,1.126,88.191,-179.1350,26.6610,0.0000
C01308=-48.976,3.143,88.238,-179.4525,26.5896,0.0000
C01309=-50.501,6.042,89.306,177.1390,25.7489,0.0000
C01310=-55.314,7.312,91.898,174.7238,24.4707,0.0000
C01311=-62.805,8.270,95.231,170.5097,20.2538,0.0000
C01312=-50.258,38.562,95.231,-159.0560,7.7820,0.0000
C01313=-44.284,33.942,91.898,-158.7700,13.5162,0.0000
C01314=-39.982,31.437,89.306,-159.3530,15.9859,0.0000
C01315=-36.853,32.408,88.238,-160.8541,18.8174,0.0000
C01316=-35.404,33.811,88.191,-160.9955,19.0754,0.0000
C01317=-34.612,34.612,88.223,-160.4524,18.5009,0.0000
C01318=-33.811,35.404,88.191,-159.9099,17.9235,0.0000
C01319=-32.408,36.854,88.238,-160.1654,18.0867,0.0000
C01320=-31.437,39.982,89.306,-162.9786,19.8146,0.0000
C01321=-33.942,44.284,91.898,-165.5396,20.6149,0.0000
C01322=-38.562,50.258,95.231,-171.6748,20.7423,0.0000
C01323=-8.270,62.805,95.231,-159.4884,-8.8986,0.0000
C01324=-7.312,55.314,91.898,-155.4374,-4.8011,0.0000
C01325=-6.042,50.501,89.306,-154.2231,-2.5767,0.0000
C01326=-3.143,48.976,88.238,-153.4094,0.4896,0.0000
C01327=-1.126,48.942,88.191,-153.3363,0.7730,0.0000
C01328=0.000,48.949,88.223,-153.3370,-0.0009,0.0000
C01329=0.000,48.503,90.377,-154.5699,-0.0008,0.0000
C01330=1.086,48.496,90.345,-154.5677,-0.7089,0.0000
C01331=3.075,48.536,90.393,-154.6411,-0.4262,0.0000
C01332=5.972,50.143,91.476,-155.4893,2.5855,0.0000
C01333=7.266,55.138,94.090,-156.8503,4.8655,0.0000
C01334=33.851,44.126,94.090,-166.6740,-19.6918,0.0000
C01335=31.234,39.679,91.476,-163.9700,-18.9626,0.0000
C01336=32.146,36.494,90.393,-161.1728,-17.3121,0.0000
C01337=33.524,35.059,90.345,-160.9177,-17.1510,0.0000
C01338=34.297,34.297,90.377,-161.4161,-17.6757,0.0000
C01339=35.059,33.525,90.345,-161.9158,-18.2040,0.0000
C01340=36.495,32.146,90.393,-161.7719,-17.9438,0.0000
C01341=39.679,31.234,91.476,-160.3279,-15.1384,0.0000
C01342=44.126,33.851,94.090,-159.8067,-12.5337,0.0000
C01343=55.138,7.266,94.090,174.7107,-23.0614,0.0000
C01344=50.143,5.972,91.476,177.1588,-24.4841,0.0000
C01345=48.536,3.075,90.393,-179.5283,-25.3581,0.0000
C01346=48.496,1.086,90.345,-179.2150,-25.4302,0.0000
C01347=48.503,0.000,90.377,-179.9991,-25.4301,0.0000
C01348=48.496,-1.085,90.345,179.2139,-25.4302,0.0000
C01349=48.536,-3.075,90.393,179.5294,-25.3580,0.0000
C01350=50.143,-5.972,91.476,-177.1585,-24.4841,0.0000
C01351=55.138,-7.266,94.090,-174.7107,-23.0616,0.0000
C01352=44.126,-33.851,94.090,159.8068,-12.5336,0.0000
C01353=39.679,-31.234,91.476,160.3281,-15.1386,0.0000
C01354=36.494,-32.146,90.393,161.7725,-17.9445,0.0000
C01355=35.059,-33.524,90.345,161.9151,-18.2032,0.0000
C01356=34.297,-34.297,90.377,161.4172,-17.6768,0.0000
C01357=33.525,-35.059,90.345,160.9169,-17.1502,0.0000
C01358=32.146,-36.495,90.393,161.1735,-17.3127,0.0000
C01359=31.234,-39.679,91.476,163.9701,-18.9628,0.0000
C01360=33.851,-44.126,94.090,166.6739,-19.6919,0.0000
C01361=7.266,-55.138,94.090,156.8503,4.8655,0.0000
C01362=5.972,-50.143,91.476,155.4893,2.5855,0.0000
C01363=3.075,-48.536,90.393,154.6411,-0.4262,0.0000
C01364=1.086,-48.496,90.345,154.5677,-0.7089,0.0000
C01365=0.000,-48.503,90.377,154.5699,-0.0008,0.0000
C01366=0.000,-48.503,90.377,154.5699,-0.0008,0.0000
C01367=-1.085,-48.496,90.345,154.5677,0.7100,0.0000
C01368=-3.075,-48.536,90.393,154.6412,0.4253,0.0000
C01369=-5.972,-50.143,91.476,155.4893,-2.5858,0.0000
C01370=-7.266,-55.138,94.090,156.8502,-4.8655,0.0000
C01371=-33.851,-44.126,94.090,166.6740,19.6918,0.0000
C01372=-31.234,-39.679,91.476,163.9700,18.9626,0.0000
C01373=-32.146,-36.494,90.393,161.1728,17.3121,0.0000
C01374=-33.524,-35.059,90.345,160.9177,17.1510,0.0000
C01375=-34.297,-34.297,90.377,161.4161,17.6757,0.0000
C01376=-35.059,-33.525,90.345,161.9158,18.2040,0.0000
C01377=-36.495,-32.146,90.393,161.7719,17.9438,0.0000
C01378=-39.679,-31.234,91.476,160.3279,15.1384,0.0000
C01379=-44.126,-33.851,94.090,159.8067,12.5337,0.0000
C01380=-55.138,-7.266,94.090,-174.7107,23.0614,0.0000
C01381=-50.143,-5.972,91.476,-177.1588,24.4841,0.0000
C01382=-48.536,-3.075,90.393,179.5283,25.3581,0.0000
C01383=-48.496,-1.086,90.345,179.2150,25.4302,0.0000
C01384=-48.503,0.000,90.377,179.9991,25.4301,0.0000
C01385=-48.496,1.085,90.345,-179.2139,25.4302,0.0000
C01386=-48.536,3.075,90.393,-179.5294,25.3580,0.0000
C01387=-50.143,5.972,91.476,177.1585,24.4841,0.0000
C01388=-55.138,7.266,94.090,174.7107,23.0616,0.0000
C01389=-44.126,33.851,94.090,-159.8068,12.5336,0.0000
C01390=-39.679,31.234,91.476,-160.3281,15.1386,0.0000
C01391=-36.494,32.146,90.393,-161.7725,17.9445,0.0000
C01392=-35.059,33.524,90.345,-161.9151,18.2032,0.0000
C01393=-34.297,34.297,90.377,-161.4172,17.6768,0.0000
C01394=-33.525,35.059,90.345,-160.9169,17.1502,0.0000
C01395=-32.146,36.495,90.393,-161.1735,17.3127,0.0000
C01396=-31.234,39.679,91.476,-163.9701,18.9628,0.0000
C01397=-33.851,44.126,94.090,-166.6739,19.6919,0.0000
C01398=-7.266,55.138,94.090,-156.8502,-4.8655,0.0000
C01399=-5.972,50.143,91.476,-155.4893,-2.5858,0.0000
C01400=-3.075,48.536,90.393,-154.6412,0.4253,0.0000
C01401=-1.085,48.496,90.345,-154.5677,0.7100,0.0000
C01402=0.000,48.503,90.377,-154.5699,-0.0008,0.0000
C01403=0.000,48.191,92.555,-155.8671,-0.0007,0.0000
C01404=1.057,48.183,92.523,-155.8635,-0.6493,0.0000
C01405=3.027,48.229,92.571,-155.9385,-0.3518,0.0000
C01406=5.927,49.917,93.664,-156.8312,2.6056,0.0000
C01407=31.106,39.488,93.664,-165.0182,-18.0631,0.0000
C01408=31.963,36.244,92.571,-162.2299,-16.4962,0.0000
C01409=33.323,34.818,92.523,-161.9634,-16.3266,0.0000
C01410=34.076,34.076,92.555,-162.4217,-16.8038,0.0000
C01411=34.818,33.324,92.523,-162.8785,-17.2865,0.0000
C01412=36.244,31.963,92.571,-162.7249,-17.0151,0.0000
C01413=39.488,31.106,93.664,-161.3445,-14.2273,0.0000
C01414=49.917,5.927,93.664,177.1661,-23.1435,0.0000
C01415=48.229,3.027,92.571,-179.6147,-24.0610,0.0000
C01416=48.183,1.057,92.523,-179.2885,-24.1348,0.0000
C01417=48.191,0.000,92.555,-179.9992,-24.1329,0.0000
C01418=48.183,-1.057,92.523,179.2875,-24.1348,0.0000
C01419=48.229,-3.027,92.571,179.6157,-24.0609,0.0000
C01420=49.918,-5.927,93.664,-177.1659,-23.1435,0.0000
C01421=39.488,-31.106,93.664,161.3446,-14.2274,0.0000
C01422=36.244,-31.963,92.571,162.7254,-17.0158,0.0000
C01423=34.818,-33.323,92.523,162.8778,-17.2858,0.0000
C01424=34.076,-34.076,92.555,162.4227,-16.8049,0.0000
C01425=33.324,-34.818,92.523,161.9628,-16.3259,0.0000
C01426=31.963,-36.244,92.571,162.2306,-16.4968,0.0000
C01427=31.106,-39.488,93.664,165.0184,-18.0633,0.0000
C01428=5.927,-49.917,93.664,156.8312,2.6056,0.0000
C01429=3.027,-48.229,92.571,155.9385,-0.3518,0.0000
C01430=1.057,-48.183,92.523,155.8635,-0.6493,0.0000
C01431=0.000,-48.191,92.555,155.8671,-0.0007,0.0000
C01432=0.000,-48.191,92.555,155.8671,-0.0007,0.0000
C01433=-1.057,-48.183,92.523,155.8635,0.6502,0.0000
C01434=-3.027,-48.229,92.571,155.9386,0.3509,0.0000
C01435=-5.927,-49.918,93.664,156.8312,-2.6059,0.0000
C01436=-31.106,-39.488,93.664,165.0182,18.0631,0.0000
C01437=-31.963,-36.244,92.571,162.2299,16.4962,0.0000
C01438=-33.323,-34.818,92.523,161.9634,16.3266,0.0000
C01439=-34.076,-34.076,92.555,162.4217,16.8038,0.0000
C01440=-34.818,-33.324,92.523,162.8785,17.2865,0.0000
C01441=-36.244,-31.963,92.571,162.7249,17.0151,0.0000
C01442=-39.488,-31.106,93.664,161.3445,14.2273,0.0000
C01443=-49.917,-5.927,93.664,-177.1661,23.1435,0.0000
C01444=-48.229,-3.027,92.571,179.6147,24.0610,0.0000
C01445=-48.183,-1.057,92.523,179.2885,24.1348,0.0000
C01446=-48.191,0.000,92.555,179.9992,24.1329,0.0000
C01447=-48.183,1.057,92.523,-179.2875,24.1348,0.0000
C01448=-48.229,3.027,92.571,-179.6157,24.0609,0.0000
C01449=-49.918,5.927,93.664,177.1659,23.1435,0.0000
C01450=-39.488,31.106,93.664,-161.3446,14.2274,0.0000
C01451=-36.244,31.963,92.571,-162.7254,17.0158,0.0000
C01452=-34.818,33.323,92.523,-162.8778,17.2858,0.0000
C01453=-34.076,34.076,92.555,-162.4227,16.8049,0.0000
C01454=-33.324,34.818,92.523,-161.9628,16.3259,0.0000
C01455=-31.963,36.244,92.571,-162.2306,16.4968,0.0000
C01456=-31.106,39.488,93.664,-165.0184,18.0633,0.0000
C01457=-5.927,49.918,93.664,-156.8312,-2.6059,0.0000
C01458=-3.027,48.229,92.571,-155.9386,0.3509,0.0000
C01459=-1.057,48.183,92.523,-155.8635,0.6502,0.0000
C01460=0.000,48.191,92.555,-155.8671,-0.0007,0.0000
C01461=0.000,48.026,94.749,-157.2267,-0.0006,0.0000
C01462=1.042,48.016,94.716,-157.2221,-0.5934,0.0000
C01463=3.002,48.067,94.764,-157.2999,-0.2669,0.0000
C01464=5.911,49.834,95.862,-158.2489,2.6368,0.0000
C01465=31.058,39.418,95.862,-166.1224,-17.1149,0.0000
C01466=31.866,36.111,94.764,-163.3344,-15.6393,0.0000
C01467=33.216,34.689,94.716,-163.0454,-15.4517,0.0000
C01468=33.959,33.959,94.749,-163.4659,-15.8848,0.0000
C01469=34.689,33.216,94.716,-163.8825,-16.3248,0.0000
C01470=36.111,31.865,94.764,-163.7101,-16.0310,0.0000
C01471=39.418,31.058,95.862,-162.4017,-13.2515,0.0000
C01472=49.834,5.911,95.862,177.1614,-21.7269,0.0000
C01473=48.067,3.002,94.764,-179.7107,-22.6998,0.0000
C01474=48.016,1.042,94.716,-179.3564,-22.7767,0.0000
C01475=48.026,0.000,94.749,-179.9993,-22.7733,0.0000
C01476=48.016,-1.041,94.716,179.3555,-22.7766,0.0000
C01477=48.067,-3.002,94.764,179.7116,-22.6997,0.0000
C01478=49.834,-5.911,95.862,-177.1611,-21.7269,0.0000
C01479=39.418,-31.058,95.862,162.4018,-13.2516,0.0000
C01480=36.111,-31.866,94.764,163.7106,-16.0316,0.0000
C01481=34.689,-33.216,94.716,163.8819,-16.3242,0.0000
C01482=33.959,-33.959,94.749,163.4668,-15.8857,0.0000
C01483=33.216,-34.689,94.716,163.0449,-15.4511,0.0000
C01484=31.865,-36.111,94.764,163.3350,-15.6399,0.0000
C01485=31.058,-39.418,95.862,166.1225,-17.1151,0.0000
C01486=5.911,-49.834,95.862,158.2489,2.6368,0.0000
C01487=3.002,-48.067,94.764,157.2999,-0.2669,0.0000
C01488=1.042,-48.016,94.716,157.2221,-0.5934,0.0000
C01489=0.000,-48.026,94.749,157.2267,-0.0006,0.0000
C01490=0.000,-48.026,94.749,157.2267,-0.0006,0.0000
C01491=-1.041,-48.016,94.716,157.2221,0.5942,0.0000
C01492=-3.002,-48.067,94.764,157.3000,0.2661,0.0000
C01493=-5.911,-49.834,95.862,158.2489,-2.6371,0.0000
C01494=-31.058,-39.418,95.862,166.1224,17.1149,0.0000
C01495=-31.866,-36.111,94.764,163.3344,15.6393,0.0000
C01496=-33.216,-34.689,94.716,163.0454,15.4517,0.0000
C01497=-33.959,-33.959,94.749,163.4659,15.8848,0.0000
C01498=-34.689,-33.216,94.716,163.8825,16.3248,0.0000
C01499=-36.111,-31.865,94.764,163.7101,16.0310,0.0000
C01500=-39.418,-31.058,95.862,162.4017,13.2515,0.0000
C01501=-49.834,-5.911,95.862,-177.1614,21.7269,0.0000
C01502=-48.067,-3.002,94.764,179.7107,22.6998,0.0000
C01503=-48.016,-1.042,94.716,179.3564,22.7767,0.0000
C01504=-48.026,0.000,94.749,179.9993,22.7733,0.0000
C01505=-48.016,1.041,94.716,-179.3555,22.7766,0.0000
C01506=-48.067,3.002,94.764,-179.7116,22.6997,0.0000
C01507=-49.834,5.911,95.862,177.1611,21.7269,0.0000
C01508=-39.418,31.058,95.862,-162.4018,13.2516,0.0000
C01509=-36.111,31.866,94.764,-163.7106,16.0316,0.0000
C01510=-34.689,33.216,94.716,-163.8819,16.3242,0.0000
C01511=-33.959,33.959,94.749,-163.4668,15.8857,0.0000
C01512=-33.216,34.689,94.716,-163.0449,15.4511,0.0000
C01513=-31.865,36.111,94.764,-163.3350,15.6399,0.0000
C01514=-31.058,39.418,95.862,-166.1225,17.1151,0.0000
C01515=-5.911,49.834,95.862,-158.2489,-2.6371,0.0000
C01516=-3.002,48.067,94.764,-157.3000,0.2661,0.0000
C01517=-1.041,48.016,94.716,-157.2221,0.5942,0.0000
C01518=0.000,48.026,94.749,-157.2267,-0.0006,0.0000
//INST
///DATE 2021/02/10 13:51
///COMM
///ATTR SC,RW,RJ
////FRAME USER 2
///GROUP1 RB1
NOP
MOVL C00000
MOVL C00001
MOVL C00002
MOVL C00003
MOVL C00004
MOVL C00005
MOVL C00006
MOVL C00007
MOVL C00008
MOVL C00009
MOVL C00010
MOVL C00011
MOVL C00012
MOVL C00013
MOVL C00014
MOVL C00015
MOVL C00016
MOVL C00017
MOVL C00018
MOVL C00019
MOVL C00020
MOVL C00021
MOVL C00022
MOVL C00023
MOVL C00024
MOVL C00025
MOVL C00026
MOVL C00027
MOVL C00028
MOVL C00029
MOVL C00030
MOVL C00031
MOVL C00032
MOVL C00033
MOVL C00034
MOVL C00035
MOVL C00036
MOVL C00037
MOVL C00038
MOVL C00039
MOVL C00040
MOVL C00041
MOVL C00042
MOVL C00043
MOVL C00044
MOVL C00045
MOVL C00046
MOVL C00047
MOVL C00048
MOVL C00049
MOVL C00050
MOVL C00051
MOVL C00052
MOVL C00053
MOVL C00054
MOVL C00055
MOVL C00056
MOVL C00057
MOVL C00058
MOVL C00059
MOVL C00060
MOVL C00061
MOVL C00062
MOVL C00063
MOVL C00064
MOVL C00065
MOVL C00066
MOVL C00067
MOVL C00068
MOVL C00069
MOVL C00070
MOVL C00071
MOVL C00072
MOVL C00073
MOVL C00074
MOVL C00075
MOVL C00076
MOVL C00077
MOVL C00078
MOVL C00079
MOVL C00080
MOVL C00081
MOVL C00082
MOVL C00083
MOVL C00084
MOVL C00085
MOVL C00086
MOVL C00087
MOVL C00088
MOVL C00089
MOVL C00090
MOVL C00091
MOVL C00092
MOVL C00093
MOVL C00094
MOVL C00095
MOVL C00096
MOVL C00097
MOVL C00098
MOVL C00099
MOVL C00100
MOVL C00101
MOVL C00102
MOVL C00103
MOVL C00104
MOVL C00105
MOVL C00106
MOVL C00107
MOVL C00108
MOVL C00109
MOVL C00110
MOVL C00111
MOVL C00112
MOVL C00113
MOVL C00114
MOVL C00115
MOVL C00116
MOVL C00117
MOVL C00118
MOVL C00119
MOVL C00120
MOVL C00121
MOVL C00122
MOVL C00123
MOVL C00124
MOVL C00125
MOVL C00126
MOVL C00127
MOVL C00128
MOVL C00129
MOVL C00130
MOVL C00131
MOVL C00132
MOVL C00133
MOVL C00134
MOVL C00135
MOVL C00136
MOVL C00137
MOVL C00138
MOVL C00139
MOVL C00140
MOVL C00141
MOVL C00142
MOVL C00143
MOVL C00144
MOVL C00145
MOVL C00146
MOVL C00147
MOVL C00148
MOVL C00149
MOVL C00150
MOVL C00151
MOVL C00152
MOVL C00153
MOVL C00154
MOVL C00155
MOVL C00156
MOVL C00157
MOVL C00158
MOVL C00159
MOVL C00160
MOVL C00161
MOVL C00162
MOVL C00163
MOVL C00164
MOVL C00165
MOVL C00166
MOVL C00167
MOVL C00168
MOVL C00169
MOVL C00170
MOVL C00171
MOVL C00172
MOVL C00173
MOVL C00174
MOVL C00175
MOVL C00176
MOVL C00177
MOVL C00178
MOVL C00179
MOVL C00180
MOVL C00181
MOVL C00182
MOVL C00183
MOVL C00184
MOVL C00185
MOVL C00186
MOVL C00187
MOVL C00188
MOVL C00189
MOVL C00190
MOVL C00191
MOVL C00192
MOVL C00193
MOVL C00194
MOVL C00195
MOVL C00196
MOVL C00197
MOVL C00198
MOVL C00199
MOVL C00200
MOVL C00201
MOVL C00202
MOVL C00203
MOVL C00204
MOVL C00205
MOVL C00206
MOVL C00207
MOVL C00208
MOVL C00209
MOVL C00210
MOVL C00211
MOVL C00212
MOVL C00213
MOVL C00214
MOVL C00215
MOVL C00216
MOVL C00217
MOVL C00218
MOVL C00219
MOVL C00220
MOVL C00221
MOVL C00222
MOVL C00223
MOVL C00224
MOVL C00225
MOVL C00226
MOVL C00227
MOVL C00228
MOVL C00229
MOVL C00230
MOVL C00231
MOVL C00232
MOVL C00233
MOVL C00234
MOVL C00235
MOVL C00236
MOVL C00237
MOVL C00238
MOVL C00239
MOVL C00240
MOVL C00241
MOVL C00242
MOVL C00243
MOVL C00244
MOVL C00245
MOVL C00246
MOVL C00247
MOVL C00248
MOVL C00249
MOVL C00250
MOVL C00251
MOVL C00252
MOVL C00253
MOVL C00254
MOVL C00255
MOVL C00256
MOVL C00257
MOVL C00258
MOVL C00259
MOVL C00260
MOVL C00261
MOVL C00262
MOVL C00263
MOVL C00264
MOVL C00265
MOVL C00266
MOVL C00267
MOVL C00268
MOVL C00269
MOVL C00270
MOVL C00271
MOVL C00272
MOVL C00273
MOVL C00274
MOVL C00275
MOVL C00276
MOVL C00277
MOVL C00278
MOVL C00279
MOVL C00280
MOVL C00281
MOVL C00282
MOVL C00283
MOVL C00284
MOVL C00285
MOVL C00286
MOVL C00287
MOVL C00288
MOVL C00289
MOVL C00290
MOVL C00291
MOVL C00292
MOVL C00293
MOVL C00294
MOVL C00295
MOVL C00296
MOVL C00297
MOVL C00298
MOVL C00299
MOVL C00300
MOVL C00301
MOVL C00302
MOVL C00303
MOVL C00304
MOVL C00305
MOVL C00306
MOVL C00307
MOVL C00308
MOVL C00309
MOVL C00310
MOVL C00311
MOVL C00312
MOVL C00313
MOVL C00314
MOVL C00315
MOVL C00316
MOVL C00317
MOVL C00318
MOVL C00319
MOVL C00320
MOVL C00321
MOVL C00322
MOVL C00323
MOVL C00324
MOVL C00325
MOVL C00326
MOVL C00327
MOVL C00328
MOVL C00329
MOVL C00330
MOVL C00331
MOVL C00332
MOVL C00333
MOVL C00334
MOVL C00335
MOVL C00336
MOVL C00337
MOVL C00338
MOVL C00339
MOVL C00340
MOVL C00341
MOVL C00342
MOVL C00343
MOVL C00344
MOVL C00345
MOVL C00346
MOVL C00347
MOVL C00348
MOVL C00349
MOVL C00350
MOVL C00351
MOVL C00352
MOVL C00353
MOVL C00354
MOVL C00355
MOVL C00356
MOVL C00357
MOVL C00358
MOVL C00359
MOVL C00360
MOVL C00361
MOVL C00362
MOVL C00363
MOVL C00364
MOVL C00365
MOVL C00366
MOVL C00367
MOVL C00368
MOVL C00369
MOVL C00370
MOVL C00371
MOVL C00372
MOVL C00373
MOVL C00374
MOVL C00375
MOVL C00376
MOVL C00377
MOVL C00378
MOVL C00379
MOVL C00380
MOVL C00381
MOVL C00382
MOVL C00383
MOVL C00384
MOVL C00385
MOVL C00386
MOVL C00387
MOVL C00388
MOVL C00389
MOVL C00390
MOVL C00391
MOVL C00392
MOVL C00393
MOVL C00394
MOVL C00395
MOVL C00396
MOVL C00397
MOVL C00398
MOVL C00399
MOVL C00400
MOVL C00401
MOVL C00402
MOVL C00403
MOVL C00404
MOVL C00405
MOVL C00406
MOVL C00407
MOVL C00408
MOVL C00409
MOVL C00410
MOVL C00411
MOVL C00412
MOVL C00413
MOVL C00414
MOVL C00415
MOVL C00416
MOVL C00417
MOVL C00418
MOVL C00419
MOVL C00420
MOVL C00421
MOVL C00422
MOVL C00423
MOVL C00424
MOVL C00425
MOVL C00426
MOVL C00427
MOVL C00428
MOVL C00429
MOVL C00430
MOVL C00431
MOVL C00432
MOVL C00433
MOVL C00434
MOVL C00435
MOVL C00436
MOVL C00437
MOVL C00438
MOVL C00439
MOVL C00440
MOVL C00441
MOVL C00442
MOVL C00443
MOVL C00444
MOVL C00445
MOVL C00446
MOVL C00447
MOVL C00448
MOVL C00449
MOVL C00450
MOVL C00451
MOVL C00452
MOVL C00453
MOVL C00454
MOVL C00455
MOVL C00456
MOVL C00457
MOVL C00458
MOVL C00459
MOVL C00460
MOVL C00461
MOVL C00462
MOVL C00463
MOVL C00464
MOVL C00465
MOVL C00466
MOVL C00467
MOVL C00468
MOVL C00469
MOVL C00470
MOVL C00471
MOVL C00472
MOVL C00473
MOVL C00474
MOVL C00475
MOVL C00476
MOVL C00477
MOVL C00478
MOVL C00479
MOVL C00480
MOVL C00481
MOVL C00482
MOVL C00483
MOVL C00484
MOVL C00485
MOVL C00486
MOVL C00487
MOVL C00488
MOVL C00489
MOVL C00490
MOVL C00491
MOVL C00492
MOVL C00493
MOVL C00494
MOVL C00495
MOVL C00496
MOVL C00497
MOVL C00498
MOVL C00499
MOVL C00500
MOVL C00501
MOVL C00502
MOVL C00503
MOVL C00504
MOVL C00505
MOVL C00506
MOVL C00507
MOVL C00508
MOVL C00509
MOVL C00510
MOVL C00511
MOVL C00512
MOVL C00513
MOVL C00514
MOVL C00515
MOVL C00516
MOVL C00517
MOVL C00518
MOVL C00519
MOVL C00520
MOVL C00521
MOVL C00522
MOVL C00523
MOVL C00524
MOVL C00525
MOVL C00526
MOVL C00527
MOVL C00528
MOVL C00529
MOVL C00530
MOVL C00531
MOVL C00532
MOVL C00533
MOVL C00534
MOVL C00535
MOVL C00536
MOVL C00537
MOVL C00538
MOVL C00539
MOVL C00540
MOVL C00541
MOVL C00542
MOVL C00543
MOVL C00544
MOVL C00545
MOVL C00546
MOVL C00547
MOVL C00548
MOVL C00549
MOVL C00550
MOVL C00551
MOVL C00552
MOVL C00553
MOVL C00554
MOVL C00555
MOVL C00556
MOVL C00557
MOVL C00558
MOVL C00559
MOVL C00560
MOVL C00561
MOVL C00562
MOVL C00563
MOVL C00564
MOVL C00565
MOVL C00566
MOVL C00567
MOVL C00568
MOVL C00569
MOVL C00570
MOVL C00571
MOVL C00572
MOVL C00573
MOVL C00574
MOVL C00575
MOVL C00576
MOVL C00577
MOVL C00578
MOVL C00579
MOVL C00580
MOVL C00581
MOVL C00582
MOVL C00583
MOVL C00584
MOVL C00585
MOVL C00586
MOVL C00587
MOVL C00588
MOVL C00589
MOVL C00590
MOVL C00591
MOVL C00592
MOVL C00593
MOVL C00594
MOVL C00595
MOVL C00596
MOVL C00597
MOVL C00598
MOVL C00599
MOVL C00600
MOVL C00601
MOVL C00602
MOVL C00603
MOVL C00604
MOVL C00605
MOVL C00606
MOVL C00607
MOVL C00608
MOVL C00609
MOVL C00610
MOVL C00611
MOVL C00612
MOVL C00613
MOVL C00614
MOVL C00615
MOVL C00616
MOVL C00617
MOVL C00618
MOVL C00619
MOVL C00620
MOVL C00621
MOVL C00622
MOVL C00623
MOVL C00624
MOVL C00625
MOVL C00626
MOVL C00627
MOVL C00628
MOVL C00629
MOVL C00630
MOVL C00631
MOVL C00632
MOVL C00633
MOVL C00634
MOVL C00635
MOVL C00636
MOVL C00637
MOVL C00638
MOVL C00639
MOVL C00640
MOVL C00641
MOVL C00642
MOVL C00643
MOVL C00644
MOVL C00645
MOVL C00646
MOVL C00647
MOVL C00648
MOVL C00649
MOVL C00650
MOVL C00651
MOVL C00652
MOVL C00653
MOVL C00654
MOVL C00655
MOVL C00656
MOVL C00657
MOVL C00658
MOVL C00659
MOVL C00660
MOVL C00661
MOVL C00662
MOVL C00663
MOVL C00664
MOVL C00665
MOVL C00666
MOVL C00667
MOVL C00668
MOVL C00669
MOVL C00670
MOVL C00671
MOVL C00672
MOVL C00673
MOVL C00674
MOVL C00675
MOVL C00676
MOVL C00677
MOVL C00678
MOVL C00679
MOVL C00680
MOVL C00681
MOVL C00682
MOVL C00683
MOVL C00684
MOVL C00685
MOVL C00686
MOVL C00687
MOVL C00688
MOVL C00689
MOVL C00690
MOVL C00691
MOVL C00692
MOVL C00693
MOVL C00694
MOVL C00695
MOVL C00696
MOVL C00697
MOVL C00698
MOVL C00699
MOVL C00700
MOVL C00701
MOVL C00702
MOVL C00703
MOVL C00704
MOVL C00705
MOVL C00706
MOVL C00707
MOVL C00708
MOVL C00709
MOVL C00710
MOVL C00711
MOVL C00712
MOVL C00713
MOVL C00714
MOVL C00715
MOVL C00716
MOVL C00717
MOVL C00718
MOVL C00719
MOVL C00720
MOVL C00721
MOVL C00722
MOVL C00723
MOVL C00724
MOVL C00725
MOVL C00726
MOVL C00727
MOVL C00728
MOVL C00729
MOVL C00730
MOVL C00731
MOVL C00732
MOVL C00733
MOVL C00734
MOVL C00735
MOVL C00736
MOVL C00737
MOVL C00738
MOVL C00739
MOVL C00740
MOVL C00741
MOVL C00742
MOVL C00743
MOVL C00744
MOVL C00745
MOVL C00746
MOVL C00747
MOVL C00748
MOVL C00749
MOVL C00750
MOVL C00751
MOVL C00752
MOVL C00753
MOVL C00754
MOVL C00755
MOVL C00756
MOVL C00757
MOVL C00758
MOVL C00759
MOVL C00760
MOVL C00761
MOVL C00762
MOVL C00763
MOVL C00764
MOVL C00765
MOVL C00766
MOVL C00767
MOVL C00768
MOVL C00769
MOVL C00770
MOVL C00771
MOVL C00772
MOVL C00773
MOVL C00774
MOVL C00775
MOVL C00776
MOVL C00777
MOVL C00778
MOVL C00779
MOVL C00780
MOVL C00781
MOVL C00782
MOVL C00783
MOVL C00784
MOVL C00785
MOVL C00786
MOVL C00787
MOVL C00788
MOVL C00789
MOVL C00790
MOVL C00791
MOVL C00792
MOVL C00793
MOVL C00794
MOVL C00795
MOVL C00796
MOVL C00797
MOVL C00798
MOVL C00799
MOVL C00800
MOVL C00801
MOVL C00802
MOVL C00803
MOVL C00804
MOVL C00805
MOVL C00806
MOVL C00807
MOVL C00808
MOVL C00809
MOVL C00810
MOVL C00811
MOVL C00812
MOVL C00813
MOVL C00814
MOVL C00815
MOVL C00816
MOVL C00817
MOVL C00818
MOVL C00819
MOVL C00820
MOVL C00821
MOVL C00822
MOVL C00823
MOVL C00824
MOVL C00825
MOVL C00826
MOVL C00827
MOVL C00828
MOVL C00829
MOVL C00830
MOVL C00831
MOVL C00832
MOVL C00833
MOVL C00834
MOVL C00835
MOVL C00836
MOVL C00837
MOVL C00838
MOVL C00839
MOVL C00840
MOVL C00841
MOVL C00842
MOVL C00843
MOVL C00844
MOVL C00845
MOVL C00846
MOVL C00847
MOVL C00848
MOVL C00849
MOVL C00850
MOVL C00851
MOVL C00852
MOVL C00853
MOVL C00854
MOVL C00855
MOVL C00856
MOVL C00857
MOVL C00858
MOVL C00859
MOVL C00860
MOVL C00861
MOVL C00862
MOVL C00863
MOVL C00864
MOVL C00865
MOVL C00866
MOVL C00867
MOVL C00868
MOVL C00869
MOVL C00870
MOVL C00871
MOVL C00872
MOVL C00873
MOVL C00874
MOVL C00875
MOVL C00876
MOVL C00877
MOVL C00878
MOVL C00879
MOVL C00880
MOVL C00881
MOVL C00882
MOVL C00883
MOVL C00884
MOVL C00885
MOVL C00886
MOVL C00887
MOVL C00888
MOVL C00889
MOVL C00890
MOVL C00891
MOVL C00892
MOVL C00893
MOVL C00894
MOVL C00895
MOVL C00896
MOVL C00897
MOVL C00898
ARCOF
MOVL C00899
ARCON
MOVL C00900
MOVL C00901
MOVL C00902
MOVL C00903
MOVL C00904
MOVL C00905
MOVL C00906
MOVL C00907
MOVL C00908
MOVL C00909
MOVL C00910
MOVL C00911
MOVL C00912
MOVL C00913
MOVL C00914
MOVL C00915
MOVL C00916
MOVL C00917
ARCOF
MOVL C00918
ARCON
MOVL C00919
MOVL C00920
MOVL C00921
MOVL C00922
MOVL C00923
MOVL C00924
MOVL C00925
MOVL C00926
MOVL C00927
MOVL C00928
MOVL C00929
MOVL C00930
MOVL C00931
MOVL C00932
MOVL C00933
MOVL C00934
MOVL C00935
MOVL C00936
ARCOF
MOVL C00937
ARCON
MOVL C00938
MOVL C00939
MOVL C00940
MOVL C00941
MOVL C00942
MOVL C00943
MOVL C00944
MOVL C00945
MOVL C00946
MOVL C00947
MOVL C00948
MOVL C00949
MOVL C00950
MOVL C00951
MOVL C00952
MOVL C00953
MOVL C00954
MOVL C00955
ARCOF
MOVL C00956
ARCON
MOVL C00957
MOVL C00958
MOVL C00959
MOVL C00960
MOVL C00961
MOVL C00962
MOVL C00963
MOVL C00964
MOVL C00965
MOVL C00966
MOVL C00967
MOVL C00968
MOVL C00969
MOVL C00970
MOVL C00971
MOVL C00972
MOVL C00973
MOVL C00974
MOVL C00975
ARCOF
MOVL C00976
ARCON
MOVL C00977
MOVL C00978
MOVL C00979
MOVL C00980
MOVL C00981
MOVL C00982
MOVL C00983
MOVL C00984
MOVL C00985
MOVL C00986
MOVL C00987
MOVL C00988
MOVL C00989
MOVL C00990
MOVL C00991
MOVL C00992
MOVL C00993
MOVL C00994
ARCOF
MOVL C00995
ARCON
MOVL C00996
MOVL C00997
MOVL C00998
MOVL C00999
MOVL C01000
MOVL C01001
MOVL C01002
MOVL C01003
MOVL C01004
MOVL C01005
MOVL C01006
MOVL C01007
MOVL C01008
MOVL C01009
MOVL C01010
MOVL C01011
MOVL C01012
MOVL C01013
ARCOF
MOVL C01014
ARCON
MOVL C01015
MOVL C01016
MOVL C01017
MOVL C01018
MOVL C01019
MOVL C01020
MOVL C01021
MOVL C01022
MOVL C01023
MOVL C01024
MOVL C01025
MOVL C01026
MOVL C01027
MOVL C01028
MOVL C01029
MOVL C01030
MOVL C01031
MOVL C01032
ARCOF
MOVL C01033
ARCON
MOVL C01034
MOVL C01035
MOVL C01036
MOVL C01037
MOVL C01038
MOVL C01039
MOVL C01040
MOVL C01041
MOVL C01042
MOVL C01043
MOVL C01044
MOVL C01045
MOVL C01046
MOVL C01047
MOVL C01048
MOVL C01049
ARCOF
MOVL C01050
ARCON
MOVL C01051
MOVL C01052
MOVL C01053
MOVL C01054
MOVL C01055
MOVL C01056
MOVL C01057
MOVL C01058
MOVL C01059
MOVL C01060
MOVL C01061
MOVL C01062
ARCOF
MOVL C01063
ARCON
MOVL C01064
MOVL C01065
MOVL C01066
MOVL C01067
MOVL C01068
MOVL C01069
MOVL C01070
MOVL C01071
MOVL C01072
MOVL C01073
MOVL C01074
MOVL C01075
ARCOF
MOVL C01076
ARCON
MOVL C01077
MOVL C01078
MOVL C01079
MOVL C01080
MOVL C01081
MOVL C01082
MOVL C01083
MOVL C01084
MOVL C01085
MOVL C01086
MOVL C01087
MOVL C01088
ARCOF
MOVL C01089
ARCON
MOVL C01090
MOVL C01091
MOVL C01092
MOVL C01093
MOVL C01094
MOVL C01095
MOVL C01096
MOVL C01097
MOVL C01098
MOVL C01099
MOVL C01100
MOVL C01101
MOVL C01102
ARCOF
MOVL C01103
ARCON
MOVL C01104
MOVL C01105
MOVL C01106
MOVL C01107
MOVL C01108
MOVL C01109
MOVL C01110
MOVL C01111
MOVL C01112
MOVL C01113
MOVL C01114
MOVL C01115
ARCOF
MOVL C01116
ARCON
MOVL C01117
MOVL C01118
MOVL C01119
MOVL C01120
MOVL C01121
MOVL C01122
MOVL C01123
MOVL C01124
MOVL C01125
MOVL C01126
MOVL C01127
MOVL C01128
ARCOF
MOVL C01129
ARCON
MOVL C01130
MOVL C01131
MOVL C01132
MOVL C01133
MOVL C01134
MOVL C01135
MOVL C01136
MOVL C01137
MOVL C01138
MOVL C01139
MOVL C01140
MOVL C01141
ARCOF
MOVL C01142
ARCON
MOVL C01143
MOVL C01144
MOVL C01145
MOVL C01146
MOVL C01147
MOVL C01148
MOVL C01149
MOVL C01150
MOVL C01151
MOVL C01152
MOVL C01153
MOVL C01154
ARCOF
MOVL C01155
ARCON
MOVL C01156
MOVL C01157
MOVL C01158
MOVL C01159
MOVL C01160
MOVL C01161
MOVL C01162
MOVL C01163
MOVL C01164
MOVL C01165
ARCOF
MOVL C01166
ARCON
MOVL C01167
MOVL C01168
MOVL C01169
MOVL C01170
MOVL C01171
MOVL C01172
MOVL C01173
MOVL C01174
MOVL C01175
MOVL C01176
ARCOF
MOVL C01177
ARCON
MOVL C01178
MOVL C01179
MOVL C01180
MOVL C01181
MOVL C01182
MOVL C01183
MOVL C01184
MOVL C01185
MOVL C01186
MOVL C01187
ARCOF
MOVL C01188
ARCON
MOVL C01189
MOVL C01190
MOVL C01191
MOVL C01192
MOVL C01193
MOVL C01194
MOVL C01195
MOVL C01196
MOVL C01197
MOVL C01198
MOVL C01199
ARCOF
MOVL C01200
ARCON
MOVL C01201
MOVL C01202
MOVL C01203
MOVL C01204
MOVL C01205
MOVL C01206
MOVL C01207
MOVL C01208
MOVL C01209
MOVL C01210
ARCOF
MOVL C01211
ARCON
MOVL C01212
MOVL C01213
MOVL C01214
MOVL C01215
MOVL C01216
MOVL C01217
MOVL C01218
MOVL C01219
MOVL C01220
MOVL C01221
ARCOF
MOVL C01222
ARCON
MOVL C01223
MOVL C01224
MOVL C01225
MOVL C01226
MOVL C01227
MOVL C01228
MOVL C01229
MOVL C01230
MOVL C01231
MOVL C01232
ARCOF
MOVL C01233
ARCON
MOVL C01234
MOVL C01235
MOVL C01236
MOVL C01237
MOVL C01238
MOVL C01239
MOVL C01240
MOVL C01241
MOVL C01242
MOVL C01243
MOVL C01244
ARCOF
MOVL C01245
ARCON
MOVL C01246
MOVL C01247
MOVL C01248
MOVL C01249
MOVL C01250
MOVL C01251
MOVL C01252
MOVL C01253
MOVL C01254
MOVL C01255
ARCOF
MOVL C01256
ARCON
MOVL C01257
MOVL C01258
MOVL C01259
MOVL C01260
MOVL C01261
MOVL C01262
MOVL C01263
MOVL C01264
MOVL C01265
MOVL C01266
ARCOF
MOVL C01267
ARCON
MOVL C01268
MOVL C01269
MOVL C01270
MOVL C01271
MOVL C01272
MOVL C01273
MOVL C01274
MOVL C01275
MOVL C01276
MOVL C01277
ARCOF
MOVL C01278
ARCON
MOVL C01279
MOVL C01280
MOVL C01281
MOVL C01282
MOVL C01283
MOVL C01284
MOVL C01285
MOVL C01286
MOVL C01287
MOVL C01288
MOVL C01289
ARCOF
MOVL C01290
ARCON
MOVL C01291
MOVL C01292
MOVL C01293
MOVL C01294
MOVL C01295
MOVL C01296
MOVL C01297
MOVL C01298
MOVL C01299
MOVL C01300
ARCOF
MOVL C01301
ARCON
MOVL C01302
MOVL C01303
MOVL C01304
MOVL C01305
MOVL C01306
MOVL C01307
MOVL C01308
MOVL C01309
MOVL C01310
MOVL C01311
ARCOF
MOVL C01312
ARCON
MOVL C01313
MOVL C01314
MOVL C01315
MOVL C01316
MOVL C01317
MOVL C01318
MOVL C01319
MOVL C01320
MOVL C01321
MOVL C01322
ARCOF
MOVL C01323
ARCON
MOVL C01324
MOVL C01325
MOVL C01326
MOVL C01327
MOVL C01328
MOVL C01329
MOVL C01330
MOVL C01331
MOVL C01332
MOVL C01333
ARCOF
MOVL C01334
ARCON
MOVL C01335
MOVL C01336
MOVL C01337
MOVL C01338
MOVL C01339
MOVL C01340
MOVL C01341
MOVL C01342
ARCOF
MOVL C01343
ARCON
MOVL C01344
MOVL C01345
MOVL C01346
MOVL C01347
MOVL C01348
MOVL C01349
MOVL C01350
MOVL C01351
ARCOF
MOVL C01352
ARCON
MOVL C01353
MOVL C01354
MOVL C01355
MOVL C01356
MOVL C01357
MOVL C01358
MOVL C01359
MOVL C01360
ARCOF
MOVL C01361
ARCON
MOVL C01362
MOVL C01363
MOVL C01364
MOVL C01365
MOVL C01366
MOVL C01367
MOVL C01368
MOVL C01369
MOVL C01370
ARCOF
MOVL C01371
ARCON
MOVL C01372
MOVL C01373
MOVL C01374
MOVL C01375
MOVL C01376
MOVL C01377
MOVL C01378
MOVL C01379
ARCOF
MOVL C01380
ARCON
MOVL C01381
MOVL C01382
MOVL C01383
MOVL C01384
MOVL C01385
MOVL C01386
MOVL C01387
MOVL C01388
ARCOF
MOVL C01389
ARCON
MOVL C01390
MOVL C01391
MOVL C01392
MOVL C01393
MOVL C01394
MOVL C01395
MOVL C01396
MOVL C01397
ARCOF
MOVL C01398
ARCON
MOVL C01399
MOVL C01400
MOVL C01401
MOVL C01402
MOVL C01403
MOVL C01404
MOVL C01405
MOVL C01406
ARCOF
MOVL C01407
ARCON
MOVL C01408
MOVL C01409
MOVL C01410
MOVL C01411
MOVL C01412
MOVL C01413
ARCOF
MOVL C01414
ARCON
MOVL C01415
MOVL C01416
MOVL C01417
MOVL C01418
MOVL C01419
MOVL C01420
ARCOF
MOVL C01421
ARCON
MOVL C01422
MOVL C01423
MOVL C01424
MOVL C01425
MOVL C01426
MOVL C01427
ARCOF
MOVL C01428
ARCON
MOVL C01429
MOVL C01430
MOVL C01431
MOVL C01432
MOVL C01433
MOVL C01434
MOVL C01435
ARCOF
MOVL C01436
ARCON
MOVL C01437
MOVL C01438
MOVL C01439
MOVL C01440
MOVL C01441
MOVL C01442
ARCOF
MOVL C01443
ARCON
MOVL C01444
MOVL C01445
MOVL C01446
MOVL C01447
MOVL C01448
MOVL C01449
ARCOF
MOVL C01450
ARCON
MOVL C01451
MOVL C01452
MOVL C01453
MOVL C01454
MOVL C01455
MOVL C01456
ARCOF
MOVL C01457
ARCON
MOVL C01458
MOVL C01459
MOVL C01460
MOVL C01461
MOVL C01462
MOVL C01463
MOVL C01464
ARCOF
MOVL C01465
ARCON
MOVL C01466
MOVL C01467
MOVL C01468
MOVL C01469
MOVL C01470
MOVL C01471
ARCOF
MOVL C01472
ARCON
MOVL C01473
MOVL C01474
MOVL C01475
MOVL C01476
MOVL C01477
MOVL C01478
ARCOF
MOVL C01479
ARCON
MOVL C01480
MOVL C01481
MOVL C01482
MOVL C01483
MOVL C01484
MOVL C01485
ARCOF
MOVL C01486
ARCON
MOVL C01487
MOVL C01488
MOVL C01489
MOVL C01490
MOVL C01491
MOVL C01492
MOVL C01493
ARCOF
MOVL C01494
ARCON
MOVL C01495
MOVL C01496
MOVL C01497
MOVL C01498
MOVL C01499
MOVL C01500
ARCOF
MOVL C01501
ARCON
MOVL C01502
MOVL C01503
MOVL C01504
MOVL C01505
MOVL C01506
MOVL C01507
ARCOF
MOVL C01508
ARCON
MOVL C01509
MOVL C01510
